LIN {X 0,Y 646.428,Z 1220.53,A -85,B 0,C 180,E1 5689.575,E2 5689.575} C_VEL
LIN {X 0,Y 649.933,Z 1168.755,A -85,B 0,C 180,E1 5694.149,E2 5694.149} C_VEL
LIN {X 0,Y 653.891,Z 1107.9,A -85,B 0,C 180,E1 5697.593,E2 5697.593} C_VEL
LIN {X 0,Y 656.115,Z 1042.809,A -85,B 0,C 180,E1 5699.566,E2 5699.566} C_VEL
LIN {X 0,Y 654.845,Z 982.129,A -85,B 0,C 180,E1 5700.484,E2 5700.484} C_VEL
LIN {X 0,Y 643.755,Z 957.34,A -85,B 0,C 180,E1 5701.335,E2 5701.335} C_VEL
LIN {X 0,Y 642.509,Z 948.94,A -85,B 0,C 180,E1 5701.958,E2 5701.958} C_VEL
LIN {X 0,Y 642.113,Z 948.94,A -85,B 0,C 180,E1 5710.571,E2 5710.571} C_VEL
LIN {X 0,Y 642.041,Z 948.94,A -85,B 0,C 180,E1 5718.158,E2 5718.158} C_VEL
LIN {X 0,Y 642.465,Z 950.207,A -85,B 0,C 180,E1 5726.456,E2 5726.456} C_VEL
LIN {X 0,Y 655.644,Z 990.43,A -85,B 0,C 180,E1 5727.732,E2 5727.732} C_VEL
LIN {X 0,Y 652.92,Z 1053.472,A -85,B 0,C 180,E1 5730.091,E2 5730.091} C_VEL
LIN {X 0,Y 649.225,Z 1112.123,A -85,B 0,C 180,E1 5733.83,E2 5733.83} C_VEL
LIN {X 0,Y 646.117,Z 1161.521,A -85,B 0,C 180,E1 5738.661,E2 5738.661} C_VEL
LIN {X 0,Y 644.175,Z 1198.737,A -85,B 0,C 180,E1 5744.292,E2 5744.292} C_VEL
LIN {X 0,Y 643.44,Z 1220.238,A -85,B 0,C 180,E1 5749.823,E2 5749.823} C_VEL
LIN {X 0,Y 643.165,Z 1229.44,A -85,B 0,C 180,E1 5755.275,E2 5755.275} C_VEL
LIN {X 0,Y 643.245,Z 1227.348,A -85,B 0,C 180,E1 5760.689,E2 5760.689} C_VEL
LIN {X 0,Y 643.485,Z 1212.675,A -85,B 0,C 180,E1 5766.446,E2 5766.446} C_VEL
LIN {X 0,Y 644.379,Z 1184.48,A -85,B 0,C 180,E1 5772.11,E2 5772.11} C_VEL
LIN {X 0,Y 646.945,Z 1142.6,A -85,B 0,C 180,E1 5777.367,E2 5777.367} C_VEL
LIN {X 0,Y 650.641,Z 1089.256,A -85,B 0,C 180,E1 5781.75,E2 5781.75} C_VEL
LIN {X 0,Y 654.328,Z 1028.717,A -85,B 0,C 180,E1 5784.935,E2 5784.935} C_VEL
LIN {X 0,Y 654.304,Z 979.292,A -85,B 0,C 180,E1 5786.611,E2 5786.611} C_VEL
LIN {X 0,Y 642.852,Z 948.94,A -85,B 0,C 180,E1 5787.961,E2 5787.961} C_VEL
LIN {X 0,Y 642.196,Z 948.94,A -85,B 0,C 180,E1 5797.622,E2 5797.622} C_VEL
LIN {X 0,Y 642.346,Z 948.94,A -85,B 0,C 180,E1 5806.13,E2 5806.13} C_VEL
LIN {X 0,Y 642.338,Z 948.94,A -85,B 0,C 180,E1 5814.631,E2 5814.631} C_VEL
LIN {X 0,Y 642.322,Z 948.94,A -85,B 0,C 180,E1 5822.535,E2 5822.535} C_VEL
LIN {X 0,Y 642.573,Z 948.94,A -85,B 0,C 180,E1 5829.943,E2 5829.943} C_VEL
LIN {X 0,Y 642.913,Z 950.765,A -85,B 0,C 180,E1 5832.35,E2 5832.35} C_VEL
LIN {X 0,Y 647.67,Z 983.205,A -85,B 0,C 180,E1 5832.85,E2 5832.85} C_VEL
LIN {X 0,Y 647.354,Z 1037.427,A -85,B 0,C 180,E1 5833.934,E2 5833.934} C_VEL
LIN {X 0,Y 645.952,Z 1082.258,A -85,B 0,C 180,E1 5836.208,E2 5836.208} C_VEL
LIN {X 0,Y 644.407,Z 1118.531,A -85,B 0,C 180,E1 5839.624,E2 5839.624} C_VEL
LIN {X 0,Y 643.495,Z 1142.198,A -85,B 0,C 180,E1 5843.876,E2 5843.876} C_VEL
LIN {X 0,Y 643.274,Z 1150.855,A -85,B 0,C 180,E1 5847.939,E2 5847.939} C_VEL
LIN {X 0,Y 643.428,Z 1148.022,A -85,B 0,C 180,E1 5851.994,E2 5851.994} C_VEL
LIN {X 0,Y 643.839,Z 1131.237,A -85,B 0,C 180,E1 5856.394,E2 5856.394} C_VEL
LIN {X 0,Y 644.983,Z 1101.717,A -85,B 0,C 180,E1 5860.128,E2 5860.128} C_VEL
LIN {X 0,Y 646.585,Z 1059.916,A -85,B 0,C 180,E1 5863.036,E2 5863.036} C_VEL
LIN {X 0,Y 647.882,Z 1011.403,A -85,B 0,C 180,E1 5864.667,E2 5864.667} C_VEL
LIN {X 0,Y 645.703,Z 960.583,A -85,B 0,C 180,E1 5865.371,E2 5865.371} C_VEL
LIN {X 0,Y 642.603,Z 948.94,A -85,B 0,C 180,E1 5865.721,E2 5865.721} C_VEL
LIN {X 0,Y 642.111,Z 948.94,A -85,B 0,C 180,E1 5872.911,E2 5872.911} C_VEL
LIN {X 0,Y 642.222,Z 948.94,A -85,B 0,C 180,E1 5880.488,E2 5880.488} C_VEL
LIN {X 0,Y 642.085,Z 948.94,A -85,B 0,C 180,E1 5888.728,E2 5888.728} C_VEL
LIN {X 0,Y 642.426,Z 948.94,A -85,B 0,C 180,E1 5896.035,E2 5896.035} C_VEL
LIN {X 0,Y 642.27,Z 948.94,A -85,B 0,C 180,E1 5904.605,E2 5904.605} C_VEL
LIN {X 0,Y 642.317,Z 948.94,A -85,B 0,C 180,E1 5912.547,E2 5912.547} C_VEL
LIN {X 0,Y 642.449,Z 948.94,A -85,B 0,C 180,E1 5919.953,E2 5919.953} C_VEL
LIN {X 0,Y 643.365,Z 948.94,A -85,B 0,C 180,E1 5928.419,E2 5928.419} C_VEL
LIN {X 0,Y 643.231,Z 948.94,A -85,B 0,C 180,E1 5937.958,E2 5937.958} C_VEL
LIN {X 0,Y 642.876,Z 948.94,A -85,B 0,C 180,E1 5946.085,E2 5946.085} C_VEL
LIN {X 0,Y 642.522,Z 948.94,A -85,B 0,C 180,E1 5954.348,E2 5954.348} C_VEL
LIN {X 0,Y 642.159,Z 948.94,A -85,B 0,C 180,E1 5962.94,E2 5962.94} C_VEL
LIN {X 0,Y 642.622,Z 948.94,A -85,B 0,C 180,E1 5970.548,E2 5970.548} C_VEL
LIN {X 0,Y 642.427,Z 948.94,A -85,B 0,C 180,E1 5979.155,E2 5979.155} C_VEL
LIN {X 0,Y 634.35,Z 948.94,A -85,B 0,C 180,E1 5982.271,E2 5982.271} C_VEL
LIN {X 0,Y 634.608,Z 948.94,A -85,B 0,C 180,E1 5990.994,E2 5990.994} C_VEL
LIN {X 0,Y 635.016,Z 950.715,A -85,B 0,C 180,E1 5996.544,E2 5996.544} C_VEL
LIN {X 0,Y 641.732,Z 974.807,A -85,B 0,C 180,E1 5998.37,E2 5998.37} C_VEL
LIN {X 0,Y 650.934,Z 992.589,A -85,B 0,C 180,E1 5999.107,E2 5999.107} C_VEL
LIN {X 0,Y 648.752,Z 1064.383,A -85,B 0,C 180,E1 6000.526,E2 6000.526} C_VEL
LIN {X 0,Y 645.117,Z 1130.85,A -85,B 0,C 180,E1 6003.225,E2 6003.225} C_VEL
LIN {X 0,Y 641.322,Z 1185.71,A -85,B 0,C 180,E1 6006.875,E2 6006.875} C_VEL
LIN {X 0,Y 638.039,Z 1233.34,A -85,B 0,C 180,E1 6011.693,E2 6011.693} C_VEL
LIN {X 0,Y 635.898,Z 1268.832,A -85,B 0,C 180,E1 6017.184,E2 6017.184} C_VEL
LIN {X 0,Y 635.105,Z 1289.609,A -85,B 0,C 180,E1 6022.548,E2 6022.548} C_VEL
LIN {X 0,Y 635.014,Z 1299.208,A -85,B 0,C 180,E1 6027.98,E2 6027.98} C_VEL
LIN {X 0,Y 634.95,Z 1297.779,A -85,B 0,C 180,E1 6033.459,E2 6033.459} C_VEL
LIN {X 0,Y 635.181,Z 1284.935,A -85,B 0,C 180,E1 6038.966,E2 6038.966} C_VEL
LIN {X 0,Y 636.236,Z 1259.453,A -85,B 0,C 180,E1 6044.536,E2 6044.536} C_VEL
LIN {X 0,Y 638.681,Z 1220.522,A -85,B 0,C 180,E1 6049.823,E2 6049.823} C_VEL
LIN {X 0,Y 642.5,Z 1168.755,A -85,B 0,C 180,E1 6054.447,E2 6054.447} C_VEL
LIN {X 0,Y 645.793,Z 1115.733,A -85,B 0,C 180,E1 6057.443,E2 6057.443} C_VEL
LIN {X 0,Y 648.319,Z 1043.871,A -85,B 0,C 180,E1 6059.711,E2 6059.711} C_VEL
LIN {X 0,Y 647.032,Z 984.427,A -85,B 0,C 180,E1 6060.682,E2 6060.682} C_VEL
LIN {X 0,Y 634.809,Z 952.48,A -85,B 0,C 180,E1 6061.606,E2 6061.606} C_VEL
LIN {X 0,Y 634.515,Z 948.94,A -85,B 0,C 180,E1 6061.902,E2 6061.902} C_VEL
LIN {X 0,Y 634.218,Z 948.94,A -85,B 0,C 180,E1 6069.387,E2 6069.387} C_VEL
LIN {X 0,Y 634.161,Z 948.94,A -85,B 0,C 180,E1 6077.009,E2 6077.009} C_VEL
LIN {X 0,Y 634.329,Z 948.94,A -85,B 0,C 180,E1 6086.148,E2 6086.148} C_VEL
LIN {X 0,Y 648.172,Z 992.693,A -85,B 0,C 180,E1 6087.529,E2 6087.529} C_VEL
LIN {X 0,Y 645.371,Z 1056.755,A -85,B 0,C 180,E1 6089.964,E2 6089.964} C_VEL
LIN {X 0,Y 641.651,Z 1112.722,A -85,B 0,C 180,E1 6093.591,E2 6093.591} C_VEL
LIN {X 0,Y 638.341,Z 1161.181,A -85,B 0,C 180,E1 6098.388,E2 6098.388} C_VEL
LIN {X 0,Y 636.325,Z 1198.539,A -85,B 0,C 180,E1 6104.093,E2 6104.093} C_VEL
LIN {X 0,Y 635.515,Z 1220.127,A -85,B 0,C 180,E1 6109.695,E2 6109.695} C_VEL
LIN {X 0,Y 635.167,Z 1229.413,A -85,B 0,C 180,E1 6115.216,E2 6115.216} C_VEL
LIN {X 0,Y 635.239,Z 1227.405,A -85,B 0,C 180,E1 6120.698,E2 6120.698} C_VEL
LIN {X 0,Y 635.5,Z 1212.876,A -85,B 0,C 180,E1 6126.508,E2 6126.508} C_VEL
LIN {X 0,Y 636.492,Z 1184.73,A -85,B 0,C 180,E1 6132.262,E2 6132.262} C_VEL
LIN {X 0,Y 639.204,Z 1143.404,A -85,B 0,C 180,E1 6137.542,E2 6137.542} C_VEL
LIN {X 0,Y 643.18,Z 1089.823,A -85,B 0,C 180,E1 6142.015,E2 6142.015} C_VEL
LIN {X 0,Y 647.176,Z 1028.483,A -85,B 0,C 180,E1 6145.268,E2 6145.268} C_VEL
LIN {X 0,Y 647.023,Z 981.257,A -85,B 0,C 180,E1 6146.902,E2 6146.902} C_VEL
LIN {X 0,Y 634.781,Z 948.94,A -85,B 0,C 180,E1 6148.335,E2 6148.335} C_VEL
LIN {X 0,Y 634.2,Z 948.94,A -85,B 0,C 180,E1 6157.627,E2 6157.627} C_VEL
LIN {X 0,Y 634.2,Z 948.94,A -85,B 0,C 180,E1 6166.966,E2 6166.966} C_VEL
LIN {X 0,Y 634.188,Z 948.94,A -85,B 0,C 180,E1 6175.749,E2 6175.749} C_VEL
LIN {X 0,Y 634.257,Z 948.94,A -85,B 0,C 180,E1 6183.848,E2 6183.848} C_VEL
LIN {X 0,Y 634.715,Z 950.059,A -85,B 0,C 180,E1 6192.111,E2 6192.111} C_VEL
LIN {X 0,Y 640.019,Z 982.816,A -85,B 0,C 180,E1 6192.638,E2 6192.638} C_VEL
LIN {X 0,Y 639.702,Z 1038.025,A -85,B 0,C 180,E1 6193.739,E2 6193.739} C_VEL
LIN {X 0,Y 638.223,Z 1083.011,A -85,B 0,C 180,E1 6196.037,E2 6196.037} C_VEL
LIN {X 0,Y 636.603,Z 1119.38,A -85,B 0,C 180,E1 6199.495,E2 6199.495} C_VEL
LIN {X 0,Y 635.609,Z 1143.099,A -85,B 0,C 180,E1 6203.799,E2 6203.799} C_VEL
LIN {X 0,Y 635.36,Z 1151.796,A -85,B 0,C 180,E1 6207.913,E2 6207.913} C_VEL
LIN {X 0,Y 635.503,Z 1149.001,A -85,B 0,C 180,E1 6212.019,E2 6212.019} C_VEL
LIN {X 0,Y 635.962,Z 1132.256,A -85,B 0,C 180,E1 6216.473,E2 6216.473} C_VEL
LIN {X 0,Y 637.199,Z 1102.796,A -85,B 0,C 180,E1 6220.253,E2 6220.253} C_VEL
LIN {X 0,Y 638.869,Z 1062.061,A -85,B 0,C 180,E1 6223.144,E2 6223.144} C_VEL
LIN {X 0,Y 640.219,Z 1013.84,A -85,B 0,C 180,E1 6224.829,E2 6224.829} C_VEL
LIN {X 0,Y 637.967,Z 961.761,A -85,B 0,C 180,E1 6225.571,E2 6225.571} C_VEL
LIN {X 0,Y 634.577,Z 948.94,A -85,B 0,C 180,E1 6225.925,E2 6225.925} C_VEL
LIN {X 0,Y 634.047,Z 948.94,A -85,B 0,C 180,E1 6233.219,E2 6233.219} C_VEL
LIN {X 0,Y 634.111,Z 948.94,A -85,B 0,C 180,E1 6240.921,E2 6240.921} C_VEL
LIN {X 0,Y 634.014,Z 948.94,A -85,B 0,C 180,E1 6249.315,E2 6249.315} C_VEL
LIN {X 0,Y 634.267,Z 948.94,A -85,B 0,C 180,E1 6256.981,E2 6256.981} C_VEL
LIN {X 0,Y 634.154,Z 948.94,A -85,B 0,C 180,E1 6265.758,E2 6265.758} C_VEL
LIN {X 0,Y 634.271,Z 948.94,A -85,B 0,C 180,E1 6273.709,E2 6273.709} C_VEL
LIN {X 0,Y 634.326,Z 948.94,A -85,B 0,C 180,E1 6281.14,E2 6281.14} C_VEL
LIN {X 0,Y 635.376,Z 948.94,A -85,B 0,C 180,E1 6288.271,E2 6288.271} C_VEL
LIN {X 0,Y 635.231,Z 948.94,A -85,B 0,C 180,E1 6297.933,E2 6297.933} C_VEL
LIN {X 0,Y 634.835,Z 948.94,A -85,B 0,C 180,E1 6306.163,E2 6306.163} C_VEL
LIN {X 0,Y 634.471,Z 948.94,A -85,B 0,C 180,E1 6314.552,E2 6314.552} C_VEL
LIN {X 0,Y 634.146,Z 948.94,A -85,B 0,C 180,E1 6322.991,E2 6322.991} C_VEL
LIN {X 0,Y 634.596,Z 948.94,A -85,B 0,C 180,E1 6330.93,E2 6330.93} C_VEL
LIN {X 0,Y 634.449,Z 948.94,A -85,B 0,C 180,E1 6339.326,E2 6339.326} C_VEL
LIN {X 0,Y 634.35,Z 948.94,A -85,B 0,C 180,E1 6342.271,E2 6342.271} C_VEL
LIN {X 0,Y 626.079,Z 948.94,A -85,B 0,C 180,E1 6345.419,E2 6345.419} C_VEL
LIN {X 0,Y 626.58,Z 948.94,A -85,B 0,C 180,E1 6354.219,E2 6354.219} C_VEL
LIN {X 0,Y 626.844,Z 950.065,A -85,B 0,C 180,E1 6356.109,E2 6356.109} C_VEL
LIN {X 0,Y 632.967,Z 973.261,A -85,B 0,C 180,E1 6357.845,E2 6357.845} C_VEL
LIN {X 0,Y 644.086,Z 995.648,A -85,B 0,C 180,E1 6358.778,E2 6358.778} C_VEL
LIN {X 0,Y 641.476,Z 1066.107,A -85,B 0,C 180,E1 6360.256,E2 6360.256} C_VEL
LIN {X 0,Y 637.418,Z 1134.053,A -85,B 0,C 180,E1 6363.134,E2 6363.134} C_VEL
LIN {X 0,Y 633.274,Z 1192.218,A -85,B 0,C 180,E1 6367.127,E2 6367.127} C_VEL
LIN {X 0,Y 629.723,Z 1239.53,A -85,B 0,C 180,E1 6372.255,E2 6372.255} C_VEL
LIN {X 0,Y 627.749,Z 1272.634,A -85,B 0,C 180,E1 6377.825,E2 6377.825} C_VEL
LIN {X 0,Y 627.021,Z 1291.733,A -85,B 0,C 180,E1 6383.228,E2 6383.228} C_VEL
LIN {X 0,Y 627.039,Z 1299.203,A -85,B 0,C 180,E1 6387.954,E2 6387.954} C_VEL
LIN {X 0,Y 626.947,Z 1297.781,A -85,B 0,C 180,E1 6393.503,E2 6393.503} C_VEL
LIN {X 0,Y 627.192,Z 1284.932,A -85,B 0,C 180,E1 6399.082,E2 6399.082} C_VEL
LIN {X 0,Y 628.329,Z 1259.448,A -85,B 0,C 180,E1 6404.723,E2 6404.723} C_VEL
LIN {X 0,Y 630.95,Z 1220.807,A -85,B 0,C 180,E1 6410.041,E2 6410.041} C_VEL
LIN {X 0,Y 634.709,Z 1171.858,A -85,B 0,C 180,E1 6414.484,E2 6414.484} C_VEL
LIN {X 0,Y 638.039,Z 1111.305,A -85,B 0,C 180,E1 6417.73,E2 6417.73} C_VEL
LIN {X 0,Y 640.739,Z 1039.901,A -85,B 0,C 180,E1 6419.968,E2 6419.968} C_VEL
LIN {X 0,Y 639.776,Z 987.462,A -85,B 0,C 180,E1 6420.86,E2 6420.86} C_VEL
LIN {X 0,Y 626.799,Z 952.316,A -85,B 0,C 180,E1 6421.684,E2 6421.684} C_VEL
LIN {X 0,Y 626.474,Z 948.94,A -85,B 0,C 180,E1 6422.081,E2 6422.081} C_VEL
LIN {X 0,Y 626.1,Z 948.94,A -85,B 0,C 180,E1 6430.236,E2 6430.236} C_VEL
LIN {X 0,Y 625.956,Z 948.94,A -85,B 0,C 180,E1 6438.197,E2 6438.197} C_VEL
LIN {X 0,Y 626.473,Z 950.495,A -85,B 0,C 180,E1 6445.907,E2 6445.907} C_VEL
LIN {X 0,Y 640.707,Z 994.789,A -85,B 0,C 180,E1 6447.317,E2 6447.317} C_VEL
LIN {X 0,Y 637.846,Z 1058.518,A -85,B 0,C 180,E1 6449.772,E2 6449.772} C_VEL
LIN {X 0,Y 634.019,Z 1114.463,A -85,B 0,C 180,E1 6453.44,E2 6453.44} C_VEL
LIN {X 0,Y 630.506,Z 1162.288,A -85,B 0,C 180,E1 6458.292,E2 6458.292} C_VEL
LIN {X 0,Y 628.438,Z 1198.34,A -85,B 0,C 180,E1 6463.888,E2 6463.888} C_VEL
LIN {X 0,Y 627.556,Z 1220.016,A -85,B 0,C 180,E1 6469.563,E2 6469.563} C_VEL
LIN {X 0,Y 627.179,Z 1229.387,A -85,B 0,C 180,E1 6475.155,E2 6475.155} C_VEL
LIN {X 0,Y 627.233,Z 1227.462,A -85,B 0,C 180,E1 6480.707,E2 6480.707} C_VEL
LIN {X 0,Y 627.527,Z 1214.163,A -85,B 0,C 180,E1 6486.262,E2 6486.262} C_VEL
LIN {X 0,Y 628.523,Z 1186.703,A -85,B 0,C 180,E1 6492.145,E2 6492.145} C_VEL
LIN {X 0,Y 631.343,Z 1146.137,A -85,B 0,C 180,E1 6497.502,E2 6497.502} C_VEL
LIN {X 0,Y 635.583,Z 1092.946,A -85,B 0,C 180,E1 6502.108,E2 6502.108} C_VEL
LIN {X 0,Y 639.779,Z 1032.03,A -85,B 0,C 180,E1 6505.451,E2 6505.451} C_VEL
LIN {X 0,Y 639.99,Z 983.789,A -85,B 0,C 180,E1 6507.174,E2 6507.174} C_VEL
LIN {X 0,Y 626.682,Z 948.94,A -85,B 0,C 180,E1 6508.707,E2 6508.707} C_VEL
LIN {X 0,Y 626.098,Z 948.94,A -85,B 0,C 180,E1 6518.201,E2 6518.201} C_VEL
LIN {X 0,Y 626.182,Z 948.94,A -85,B 0,C 180,E1 6526.278,E2 6526.278} C_VEL
LIN {X 0,Y 626.19,Z 948.94,A -85,B 0,C 180,E1 6535.249,E2 6535.249} C_VEL
LIN {X 0,Y 626.255,Z 948.94,A -85,B 0,C 180,E1 6543.333,E2 6543.333} C_VEL
LIN {X 0,Y 626.611,Z 948.94,A -85,B 0,C 180,E1 6551.857,E2 6551.857} C_VEL
LIN {X 0,Y 632.346,Z 981.432,A -85,B 0,C 180,E1 6552.409,E2 6552.409} C_VEL
LIN {X 0,Y 632.084,Z 1037.191,A -85,B 0,C 180,E1 6553.492,E2 6553.492} C_VEL
LIN {X 0,Y 630.585,Z 1082.539,A -85,B 0,C 180,E1 6555.776,E2 6555.776} C_VEL
LIN {X 0,Y 628.926,Z 1118.829,A -85,B 0,C 180,E1 6559.189,E2 6559.189} C_VEL
LIN {X 0,Y 627.934,Z 1142.695,A -85,B 0,C 180,E1 6563.375,E2 6563.375} C_VEL
LIN {X 0,Y 627.434,Z 1152.737,A -85,B 0,C 180,E1 6567.887,E2 6567.887} C_VEL
LIN {X 0,Y 627.592,Z 1149.978,A -85,B 0,C 180,E1 6572.044,E2 6572.044} C_VEL
LIN {X 0,Y 628.079,Z 1133.276,A -85,B 0,C 180,E1 6576.555,E2 6576.555} C_VEL
LIN {X 0,Y 629.416,Z 1103.874,A -85,B 0,C 180,E1 6580.381,E2 6580.381} C_VEL
LIN {X 0,Y 631.176,Z 1062.572,A -85,B 0,C 180,E1 6583.343,E2 6583.343} C_VEL
LIN {X 0,Y 632.576,Z 1015.377,A -85,B 0,C 180,E1 6585.012,E2 6585.012} C_VEL
LIN {X 0,Y 630.22,Z 962.615,A -85,B 0,C 180,E1 6585.781,E2 6585.781} C_VEL
LIN {X 0,Y 626.541,Z 948.94,A -85,B 0,C 180,E1 6586.134,E2 6586.134} C_VEL
LIN {X 0,Y 625.957,Z 948.94,A -85,B 0,C 180,E1 6594.56,E2 6594.56} C_VEL
LIN {X 0,Y 626.037,Z 948.94,A -85,B 0,C 180,E1 6601.364,E2 6601.364} C_VEL
LIN {X 0,Y 625.922,Z 948.94,A -85,B 0,C 180,E1 6609.924,E2 6609.924} C_VEL
LIN {X 0,Y 626.144,Z 948.94,A -85,B 0,C 180,E1 6618.175,E2 6618.175} C_VEL
LIN {X 0,Y 626.16,Z 948.94,A -85,B 0,C 180,E1 6626.932,E2 6626.932} C_VEL
LIN {X 0,Y 626.41,Z 948.94,A -85,B 0,C 180,E1 6635.191,E2 6635.191} C_VEL
LIN {X 0,Y 626.674,Z 948.94,A -85,B 0,C 180,E1 6643.813,E2 6643.813} C_VEL
LIN {X 0,Y 626.802,Z 948.94,A -85,B 0,C 180,E1 6650.93,E2 6650.93} C_VEL
LIN {X 0,Y 627.241,Z 948.94,A -85,B 0,C 180,E1 6657.906,E2 6657.906} C_VEL
LIN {X 0,Y 626.804,Z 948.94,A -85,B 0,C 180,E1 6666.242,E2 6666.242} C_VEL
LIN {X 0,Y 626.438,Z 948.94,A -85,B 0,C 180,E1 6674.724,E2 6674.724} C_VEL
LIN {X 0,Y 626.313,Z 948.94,A -85,B 0,C 180,E1 6682.048,E2 6682.048} C_VEL
LIN {X 0,Y 626.574,Z 948.94,A -85,B 0,C 180,E1 6691.371,E2 6691.371} C_VEL
LIN {X 0,Y 626.387,Z 948.94,A -85,B 0,C 180,E1 6699.933,E2 6699.933} C_VEL
LIN {X 0,Y 626.079,Z 948.94,A -85,B 0,C 180,E1 6705.419,E2 6705.419} C_VEL
LIN {X 0,Y 618.251,Z 948.94,A -85,B 0,C 180,E1 6708.612,E2 6708.612} C_VEL
LIN {X 0,Y 618.915,Z 950.77,A -85,B 0,C 180,E1 6715.779,E2 6715.779} C_VEL
LIN {X 0,Y 624.625,Z 971.408,A -85,B 0,C 180,E1 6717.323,E2 6717.323} C_VEL
LIN {X 0,Y 637.204,Z 1000.02,A -85,B 0,C 180,E1 6718.456,E2 6718.456} C_VEL
LIN {X 0,Y 634.063,Z 1071.337,A -85,B 0,C 180,E1 6720.099,E2 6720.099} C_VEL
LIN {X 0,Y 629.657,Z 1138.218,A -85,B 0,C 180,E1 6723.096,E2 6723.096} C_VEL
LIN {X 0,Y 625.202,Z 1196.624,A -85,B 0,C 180,E1 6727.288,E2 6727.288} C_VEL
LIN {X 0,Y 621.925,Z 1239.976,A -85,B 0,C 180,E1 6732.085,E2 6732.085} C_VEL
LIN {X 0,Y 619.805,Z 1272.628,A -85,B 0,C 180,E1 6737.667,E2 6737.667} C_VEL
LIN {X 0,Y 619.05,Z 1291.611,A -85,B 0,C 180,E1 6743.096,E2 6743.096} C_VEL
LIN {X 0,Y 619.045,Z 1299.198,A -85,B 0,C 180,E1 6747.928,E2 6747.928} C_VEL
LIN {X 0,Y 618.943,Z 1297.777,A -85,B 0,C 180,E1 6753.548,E2 6753.548} C_VEL
LIN {X 0,Y 619.237,Z 1284.93,A -85,B 0,C 180,E1 6759.199,E2 6759.199} C_VEL
LIN {X 0,Y 620.438,Z 1259.444,A -85,B 0,C 180,E1 6764.915,E2 6764.915} C_VEL
LIN {X 0,Y 623.332,Z 1219.873,A -85,B 0,C 180,E1 6770.408,E2 6770.408} C_VEL
LIN {X 0,Y 626.61,Z 1175.783,A -85,B 0,C 180,E1 6774.299,E2 6774.299} C_VEL
LIN {X 0,Y 630.082,Z 1112.795,A -85,B 0,C 180,E1 6777.787,E2 6777.787} C_VEL
LIN {X 0,Y 633.027,Z 1038.375,A -85,B 0,C 180,E1 6780.182,E2 6780.182} C_VEL
LIN {X 0,Y 632.053,Z 989.56,A -85,B 0,C 180,E1 6781.066,E2 6781.066} C_VEL
LIN {X 0,Y 619.47,Z 954.539,A -85,B 0,C 180,E1 6781.911,E2 6781.911} C_VEL
LIN {X 0,Y 618.455,Z 948.94,A -85,B 0,C 180,E1 6782.172,E2 6782.172} C_VEL
LIN {X 0,Y 618.077,Z 948.94,A -85,B 0,C 180,E1 6790.627,E2 6790.627} C_VEL
LIN {X 0,Y 617.935,Z 948.94,A -85,B 0,C 180,E1 6798.547,E2 6798.547} C_VEL
LIN {X 0,Y 618.365,Z 949.669,A -85,B 0,C 180,E1 6805.599,E2 6805.599} C_VEL
LIN {X 0,Y 633.261,Z 997.105,A -85,B 0,C 180,E1 6807.107,E2 6807.107} C_VEL
LIN {X 0,Y 630.352,Z 1059.6,A -85,B 0,C 180,E1 6809.541,E2 6809.541} C_VEL
LIN {X 0,Y 626.359,Z 1116.16,A -85,B 0,C 180,E1 6813.292,E2 6813.292} C_VEL
LIN {X 0,Y 622.674,Z 1163.395,A -85,B 0,C 180,E1 6818.193,E2 6818.193} C_VEL
LIN {X 0,Y 620.378,Z 1199.846,A -85,B 0,C 180,E1 6824.038,E2 6824.038} C_VEL
LIN {X 0,Y 619.335,Z 1221.829,A -85,B 0,C 180,E1 6830.136,E2 6830.136} C_VEL
LIN {X 0,Y 619.179,Z 1229.36,A -85,B 0,C 180,E1 6835.092,E2 6835.092} C_VEL
LIN {X 0,Y 619.228,Z 1227.518,A -85,B 0,C 180,E1 6840.716,E2 6840.716} C_VEL
LIN {X 0,Y 619.526,Z 1212.665,A -85,B 0,C 180,E1 6846.815,E2 6846.815} C_VEL
LIN {X 0,Y 620.684,Z 1185.427,A -85,B 0,C 180,E1 6852.549,E2 6852.549} C_VEL
LIN {X 0,Y 623.724,Z 1144.944,A -85,B 0,C 180,E1 6857.901,E2 6857.901} C_VEL
LIN {X 0,Y 628.258,Z 1092.305,A -85,B 0,C 180,E1 6862.473,E2 6862.473} C_VEL
LIN {X 0,Y 632.699,Z 1031.07,A -85,B 0,C 180,E1 6865.83,E2 6865.83} C_VEL
LIN {X 0,Y 632.951,Z 986.353,A -85,B 0,C 180,E1 6867.452,E2 6867.452} C_VEL
LIN {X 0,Y 618.528,Z 948.94,A -85,B 0,C 180,E1 6869.237,E2 6869.237} C_VEL
LIN {X 0,Y 618.144,Z 948.94,A -85,B 0,C 180,E1 6877.029,E2 6877.029} C_VEL
LIN {X 0,Y 618.174,Z 948.94,A -85,B 0,C 180,E1 6886.432,E2 6886.432} C_VEL
LIN {X 0,Y 618.192,Z 948.94,A -85,B 0,C 180,E1 6895.36,E2 6895.36} C_VEL
LIN {X 0,Y 618.254,Z 948.94,A -85,B 0,C 180,E1 6903.677,E2 6903.677} C_VEL
LIN {X 0,Y 618.771,Z 950.635,A -85,B 0,C 180,E1 6911.648,E2 6911.648} C_VEL
LIN {X 0,Y 624.724,Z 982.863,A -85,B 0,C 180,E1 6912.209,E2 6912.209} C_VEL
LIN {X 0,Y 624.437,Z 1038.371,A -85,B 0,C 180,E1 6913.308,E2 6913.308} C_VEL
LIN {X 0,Y 622.867,Z 1083.29,A -85,B 0,C 180,E1 6915.596,E2 6915.596} C_VEL
LIN {X 0,Y 621.131,Z 1119.667,A -85,B 0,C 180,E1 6919.052,E2 6919.052} C_VEL
LIN {X 0,Y 620.039,Z 1143.673,A -85,B 0,C 180,E1 6923.311,E2 6923.311} C_VEL
LIN {X 0,Y 619.52,Z 1153.678,A -85,B 0,C 180,E1 6927.86,E2 6927.86} C_VEL
LIN {X 0,Y 619.665,Z 1150.957,A -85,B 0,C 180,E1 6932.07,E2 6932.07} C_VEL
LIN {X 0,Y 620.206,Z 1134.293,A -85,B 0,C 180,E1 6936.638,E2 6936.638} C_VEL
LIN {X 0,Y 621.646,Z 1104.95,A -85,B 0,C 180,E1 6940.513,E2 6940.513} C_VEL
LIN {X 0,Y 623.493,Z 1063.739,A -85,B 0,C 180,E1 6943.51,E2 6943.51} C_VEL
LIN {X 0,Y 624.931,Z 1016.15,A -85,B 0,C 180,E1 6945.215,E2 6945.215} C_VEL
LIN {X 0,Y 622.549,Z 963.94,A -85,B 0,C 180,E1 6945.987,E2 6945.987} C_VEL
LIN {X 0,Y 618.515,Z 948.94,A -85,B 0,C 180,E1 6946.35,E2 6946.35} C_VEL
LIN {X 0,Y 617.962,Z 948.94,A -85,B 0,C 180,E1 6953.861,E2 6953.861} C_VEL
LIN {X 0,Y 617.955,Z 948.94,A -85,B 0,C 180,E1 6962.046,E2 6962.046} C_VEL
LIN {X 0,Y 617.897,Z 948.94,A -85,B 0,C 180,E1 6970.55,E2 6970.55} C_VEL
LIN {X 0,Y 618.146,Z 948.94,A -85,B 0,C 180,E1 6978.42,E2 6978.42} C_VEL
LIN {X 0,Y 618.157,Z 948.94,A -85,B 0,C 180,E1 6986.448,E2 6986.448} C_VEL
LIN {X 0,Y 618.303,Z 948.94,A -85,B 0,C 180,E1 6994.543,E2 6994.543} C_VEL
LIN {X 0,Y 618.637,Z 948.94,A -85,B 0,C 180,E1 7003.597,E2 7003.597} C_VEL
LIN {X 0,Y 618.846,Z 948.94,A -85,B 0,C 180,E1 7010.813,E2 7010.813} C_VEL
LIN {X 0,Y 619.24,Z 948.94,A -85,B 0,C 180,E1 7017.879,E2 7017.879} C_VEL
LIN {X 0,Y 618.58,Z 948.94,A -85,B 0,C 180,E1 7026.886,E2 7026.886} C_VEL
LIN {X 0,Y 618.388,Z 948.94,A -85,B 0,C 180,E1 7034.92,E2 7034.92} C_VEL
LIN {X 0,Y 618.1,Z 948.94,A -85,B 0,C 180,E1 7043.086,E2 7043.086} C_VEL
LIN {X 0,Y 618.517,Z 948.94,A -85,B 0,C 180,E1 7051.827,E2 7051.827} C_VEL
LIN {X 0,Y 618.376,Z 948.94,A -85,B 0,C 180,E1 7060.557,E2 7060.557} C_VEL
LIN {X 0,Y 618.251,Z 948.94,A -85,B 0,C 180,E1 7068.612,E2 7068.612} C_VEL
LIN {X 0,Y 610.423,Z 948.94,A -85,B 0,C 180,E1 7071.854,E2 7071.854} C_VEL
LIN {X 0,Y 610.931,Z 950.999,A -85,B 0,C 180,E1 7075.398,E2 7075.398} C_VEL
LIN {X 0,Y 616.423,Z 969.525,A -85,B 0,C 180,E1 7076.791,E2 7076.791} C_VEL
LIN {X 0,Y 630.273,Z 1003.491,A -85,B 0,C 180,E1 7078.131,E2 7078.131} C_VEL
LIN {X 0,Y 626.759,Z 1074.429,A -85,B 0,C 180,E1 7079.874,E2 7079.874} C_VEL
LIN {X 0,Y 621.981,Z 1140.429,A -85,B 0,C 180,E1 7082.959,E2 7082.959} C_VEL
LIN {X 0,Y 617.26,Z 1198.745,A -85,B 0,C 180,E1 7087.284,E2 7087.284} C_VEL
LIN {X 0,Y 613.915,Z 1242.494,A -85,B 0,C 180,E1 7092.209,E2 7092.209} C_VEL
LIN {X 0,Y 611.772,Z 1274.278,A -85,B 0,C 180,E1 7097.866,E2 7097.866} C_VEL
LIN {X 0,Y 610.988,Z 1292.968,A -85,B 0,C 180,E1 7103.619,E2 7103.619} C_VEL
LIN {X 0,Y 610.897,Z 1299.825,A -85,B 0,C 180,E1 7109.324,E2 7109.324} C_VEL
LIN {X 0,Y 611.028,Z 1295.691,A -85,B 0,C 180,E1 7115.021,E2 7115.021} C_VEL
LIN {X 0,Y 611.898,Z 1277.935,A -85,B 0,C 180,E1 7121.247,E2 7121.247} C_VEL
LIN {X 0,Y 614,Z 1245.824,A -85,B 0,C 180,E1 7127.286,E2 7127.286} C_VEL
LIN {X 0,Y 616.497,Z 1208.513,A -85,B 0,C 180,E1 7131.702,E2 7131.702} C_VEL
LIN {X 0,Y 619.944,Z 1153.925,A -85,B 0,C 180,E1 7135.787,E2 7135.787} C_VEL
LIN {X 0,Y 623.434,Z 1085.707,A -85,B 0,C 180,E1 7138.975,E2 7138.975} C_VEL
LIN {X 0,Y 626.162,Z 1007.58,A -85,B 0,C 180,E1 7140.976,E2 7140.976} C_VEL
LIN {X 0,Y 623.591,Z 990.18,A -85,B 0,C 180,E1 7141.323,E2 7141.323} C_VEL
LIN {X 0,Y 610.42,Z 948.94,A -85,B 0,C 180,E1 7142.345,E2 7142.345} C_VEL
LIN {X 0,Y 610.079,Z 948.94,A -85,B 0,C 180,E1 7151.275,E2 7151.275} C_VEL
LIN {X 0,Y 609.921,Z 948.94,A -85,B 0,C 180,E1 7159.406,E2 7159.406} C_VEL
LIN {X 0,Y 610.447,Z 950.512,A -85,B 0,C 180,E1 7165.306,E2 7165.306} C_VEL
LIN {X 0,Y 625.776,Z 1000.068,A -85,B 0,C 180,E1 7166.908,E2 7166.908} C_VEL
LIN {X 0,Y 622.717,Z 1063.063,A -85,B 0,C 180,E1 7169.432,E2 7169.432} C_VEL
LIN {X 0,Y 618.644,Z 1118.961,A -85,B 0,C 180,E1 7173.236,E2 7173.236} C_VEL
LIN {X 0,Y 614.856,Z 1164.474,A -85,B 0,C 180,E1 7178.086,E2 7178.086} C_VEL
LIN {X 0,Y 612.499,Z 1199.646,A -85,B 0,C 180,E1 7183.827,E2 7183.827} C_VEL
LIN {X 0,Y 611.382,Z 1221.73,A -85,B 0,C 180,E1 7190.006,E2 7190.006} C_VEL
LIN {X 0,Y 611.176,Z 1229.325,A -85,B 0,C 180,E1 7195.028,E2 7195.028} C_VEL
LIN {X 0,Y 611.224,Z 1227.573,A -85,B 0,C 180,E1 7200.725,E2 7200.725} C_VEL
LIN {X 0,Y 611.536,Z 1213.247,A -85,B 0,C 180,E1 7206.773,E2 7206.773} C_VEL
LIN {X 0,Y 612.83,Z 1185.677,A -85,B 0,C 180,E1 7212.712,E2 7212.712} C_VEL
LIN {X 0,Y 616.166,Z 1143.96,A -85,B 0,C 180,E1 7218.307,E2 7218.307} C_VEL
LIN {X 0,Y 621.042,Z 1090.403,A -85,B 0,C 180,E1 7222.939,E2 7222.939} C_VEL
LIN {X 0,Y 625.784,Z 1028.143,A -85,B 0,C 180,E1 7226.301,E2 7226.301} C_VEL
LIN {X 0,Y 625.691,Z 988.359,A -85,B 0,C 180,E1 7227.756,E2 7227.756} C_VEL
LIN {X 0,Y 610.39,Z 948.94,A -85,B 0,C 180,E1 7229.635,E2 7229.635} C_VEL
LIN {X 0,Y 609.985,Z 948.94,A -85,B 0,C 180,E1 7238.359,E2 7238.359} C_VEL
LIN {X 0,Y 610.144,Z 948.94,A -85,B 0,C 180,E1 7247.23,E2 7247.23} C_VEL
LIN {X 0,Y 610.157,Z 948.94,A -85,B 0,C 180,E1 7255.936,E2 7255.936} C_VEL
LIN {X 0,Y 610.264,Z 948.94,A -85,B 0,C 180,E1 7264.17,E2 7264.17} C_VEL
LIN {X 0,Y 610.807,Z 950.847,A -85,B 0,C 180,E1 7271.404,E2 7271.404} C_VEL
LIN {X 0,Y 617.069,Z 981.887,A -85,B 0,C 180,E1 7271.971,E2 7271.971} C_VEL
LIN {X 0,Y 616.827,Z 1038.25,A -85,B 0,C 180,E1 7273.072,E2 7273.072} C_VEL
LIN {X 0,Y 615.178,Z 1084.052,A -85,B 0,C 180,E1 7275.412,E2 7275.412} C_VEL
LIN {X 0,Y 613.342,Z 1120.506,A -85,B 0,C 180,E1 7278.911,E2 7278.911} C_VEL
LIN {X 0,Y 612.256,Z 1143.851,A -85,B 0,C 180,E1 7283.033,E2 7283.033} C_VEL
LIN {X 0,Y 611.597,Z 1154.619,A -85,B 0,C 180,E1 7287.832,E2 7287.832} C_VEL
LIN {X 0,Y 611.728,Z 1151.938,A -85,B 0,C 180,E1 7292.097,E2 7292.097} C_VEL
LIN {X 0,Y 612.342,Z 1135.601,A -85,B 0,C 180,E1 7296.668,E2 7296.668} C_VEL
LIN {X 0,Y 613.872,Z 1106.025,A -85,B 0,C 180,E1 7300.647,E2 7300.647} C_VEL
LIN {X 0,Y 615.805,Z 1064.885,A -85,B 0,C 180,E1 7303.682,E2 7303.682} C_VEL
LIN {X 0,Y 617.274,Z 1017.605,A -85,B 0,C 180,E1 7305.409,E2 7305.409} C_VEL
LIN {X 0,Y 615.138,Z 966.152,A -85,B 0,C 180,E1 7306.179,E2 7306.179} C_VEL
LIN {X 0,Y 610.488,Z 948.94,A -85,B 0,C 180,E1 7306.571,E2 7306.571} C_VEL
LIN {X 0,Y 609.915,Z 948.94,A -85,B 0,C 180,E1 7314.692,E2 7314.692} C_VEL
LIN {X 0,Y 609.942,Z 948.94,A -85,B 0,C 180,E1 7322.29,E2 7322.29} C_VEL
LIN {X 0,Y 609.912,Z 948.94,A -85,B 0,C 180,E1 7331.195,E2 7331.195} C_VEL
LIN {X 0,Y 610.117,Z 948.94,A -85,B 0,C 180,E1 7339.277,E2 7339.277} C_VEL
LIN {X 0,Y 610.218,Z 948.94,A -85,B 0,C 180,E1 7347.655,E2 7347.655} C_VEL
LIN {X 0,Y 610.39,Z 948.94,A -85,B 0,C 180,E1 7355.762,E2 7355.762} C_VEL
LIN {X 0,Y 610.898,Z 948.94,A -85,B 0,C 180,E1 7364.863,E2 7364.863} C_VEL
LIN {X 0,Y 610.475,Z 948.94,A -85,B 0,C 180,E1 7372.126,E2 7372.126} C_VEL
LIN {X 0,Y 610.627,Z 948.94,A -85,B 0,C 180,E1 7379.274,E2 7379.274} C_VEL
LIN {X 0,Y 610.731,Z 948.94,A -85,B 0,C 180,E1 7386.407,E2 7386.407} C_VEL
LIN {X 0,Y 610.329,Z 948.94,A -85,B 0,C 180,E1 7395.122,E2 7395.122} C_VEL
LIN {X 0,Y 610.169,Z 948.94,A -85,B 0,C 180,E1 7402.664,E2 7402.664} C_VEL
LIN {X 0,Y 610.481,Z 948.94,A -85,B 0,C 180,E1 7411.037,E2 7411.037} C_VEL
LIN {X 0,Y 610.338,Z 948.94,A -85,B 0,C 180,E1 7419.338,E2 7419.338} C_VEL
LIN {X 0,Y 610.278,Z 948.94,A -85,B 0,C 180,E1 7428.835,E2 7428.835} C_VEL
LIN {X 0,Y 610.423,Z 948.94,A -85,B 0,C 180,E1 7431.854,E2 7431.854} C_VEL
LIN {X 0,Y 602.479,Z 948.94,A -85,B 0,C 180,E1 7433.992,E2 7433.992} C_VEL
LIN {X 0,Y 602.677,Z 950.167,A -85,B 0,C 180,E1 7434.91,E2 7434.91} C_VEL
LIN {X 0,Y 608.326,Z 968.385,A -85,B 0,C 180,E1 7436.26,E2 7436.26} C_VEL
LIN {X 0,Y 623.414,Z 1005.825,A -85,B 0,C 180,E1 7437.786,E2 7437.786} C_VEL
LIN {X 0,Y 619.57,Z 1074.847,A -85,B 0,C 180,E1 7439.552,E2 7439.552} C_VEL
LIN {X 0,Y 614.349,Z 1141.966,A -85,B 0,C 180,E1 7442.778,E2 7442.778} C_VEL
LIN {X 0,Y 609.386,Z 1200.193,A -85,B 0,C 180,E1 7447.218,E2 7447.218} C_VEL
LIN {X 0,Y 605.833,Z 1245.168,A -85,B 0,C 180,E1 7452.423,E2 7452.423} C_VEL
LIN {X 0,Y 603.779,Z 1275.64,A -85,B 0,C 180,E1 7458.013,E2 7458.013} C_VEL
LIN {X 0,Y 603,Z 1293.346,A -85,B 0,C 180,E1 7463.722,E2 7463.722} C_VEL
LIN {X 0,Y 602.898,Z 1299.822,A -85,B 0,C 180,E1 7469.315,E2 7469.315} C_VEL
LIN {X 0,Y 603.049,Z 1295.695,A -85,B 0,C 180,E1 7475.088,E2 7475.088} C_VEL
LIN {X 0,Y 603.996,Z 1277.931,A -85,B 0,C 180,E1 7481.397,E2 7481.397} C_VEL
LIN {X 0,Y 606.04,Z 1247.08,A -85,B 0,C 180,E1 7487.293,E2 7487.293} C_VEL
LIN {X 0,Y 609.012,Z 1202.729,A -85,B 0,C 180,E1 7492.271,E2 7492.271} C_VEL
LIN {X 0,Y 612.488,Z 1146.505,A -85,B 0,C 180,E1 7496.299,E2 7496.299} C_VEL
LIN {X 0,Y 615.915,Z 1076.981,A -85,B 0,C 180,E1 7499.424,E2 7499.424} C_VEL
LIN {X 0,Y 617.847,Z 996.189,A -85,B 0,C 180,E1 7501.413,E2 7501.413} C_VEL
LIN {X 0,Y 604.874,Z 958.099,A -85,B 0,C 180,E1 7502.415,E2 7502.415} C_VEL
LIN {X 0,Y 602.302,Z 948.94,A -85,B 0,C 180,E1 7502.836,E2 7502.836} C_VEL
LIN {X 0,Y 602.043,Z 948.94,A -85,B 0,C 180,E1 7511.972,E2 7511.972} C_VEL
LIN {X 0,Y 601.954,Z 948.94,A -85,B 0,C 180,E1 7520.3,E2 7520.3} C_VEL
LIN {X 0,Y 602.494,Z 950.806,A -85,B 0,C 180,E1 7524.992,E2 7524.992} C_VEL
LIN {X 0,Y 618.32,Z 1002.184,A -85,B 0,C 180,E1 7526.68,E2 7526.68} C_VEL
LIN {X 0,Y 615.17,Z 1065.212,A -85,B 0,C 180,E1 7529.249,E2 7529.249} C_VEL
LIN {X 0,Y 611.034,Z 1119.915,A -85,B 0,C 180,E1 7533.026,E2 7533.026} C_VEL
LIN {X 0,Y 607.027,Z 1166.152,A -85,B 0,C 180,E1 7538.027,E2 7538.027} C_VEL
LIN {X 0,Y 604.445,Z 1201.152,A -85,B 0,C 180,E1 7543.98,E2 7543.98} C_VEL
LIN {X 0,Y 603.45,Z 1221.624,A -85,B 0,C 180,E1 7549.874,E2 7549.874} C_VEL
LIN {X 0,Y 603.173,Z 1229.285,A -85,B 0,C 180,E1 7554.961,E2 7554.961} C_VEL
LIN {X 0,Y 603.22,Z 1227.627,A -85,B 0,C 180,E1 7560.735,E2 7560.735} C_VEL
LIN {X 0,Y 603.56,Z 1213.339,A -85,B 0,C 180,E1 7566.875,E2 7566.875} C_VEL
LIN {X 0,Y 604.946,Z 1185.959,A -85,B 0,C 180,E1 7572.881,E2 7572.881} C_VEL
LIN {X 0,Y 608.399,Z 1146.119,A -85,B 0,C 180,E1 7578.367,E2 7578.367} C_VEL
LIN {X 0,Y 613.482,Z 1093.229,A -85,B 0,C 180,E1 7583.069,E2 7583.069} C_VEL
LIN {X 0,Y 618.396,Z 1032.11,A -85,B 0,C 180,E1 7586.485,E2 7586.485} C_VEL
LIN {X 0,Y 618.784,Z 991.312,A -85,B 0,C 180,E1 7588.021,E2 7588.021} C_VEL
LIN {X 0,Y 602.285,Z 948.94,A -85,B 0,C 180,E1 7590.074,E2 7590.074} C_VEL
LIN {X 0,Y 601.991,Z 948.94,A -85,B 0,C 180,E1 7598.168,E2 7598.168} C_VEL
LIN {X 0,Y 602.103,Z 948.94,A -85,B 0,C 180,E1 7606.084,E2 7606.084} C_VEL
LIN {X 0,Y 602.113,Z 948.94,A -85,B 0,C 180,E1 7615.035,E2 7615.035} C_VEL
LIN {X 0,Y 602.219,Z 948.94,A -85,B 0,C 180,E1 7623.799,E2 7623.799} C_VEL
LIN {X 0,Y 602.623,Z 950.198,A -85,B 0,C 180,E1 7631.134,E2 7631.134} C_VEL
LIN {X 0,Y 609.485,Z 982.889,A -85,B 0,C 180,E1 7631.752,E2 7631.752} C_VEL
LIN {X 0,Y 609.162,Z 1040.383,A -85,B 0,C 180,E1 7632.906,E2 7632.906} C_VEL
LIN {X 0,Y 607.396,Z 1086.061,A -85,B 0,C 180,E1 7635.313,E2 7635.313} C_VEL
LIN {X 0,Y 605.388,Z 1122.804,A -85,B 0,C 180,E1 7638.951,E2 7638.951} C_VEL
LIN {X 0,Y 604.058,Z 1146.706,A -85,B 0,C 180,E1 7643.474,E2 7643.474} C_VEL
LIN {X 0,Y 603.682,Z 1155.56,A -85,B 0,C 180,E1 7647.804,E2 7647.804} C_VEL
LIN {X 0,Y 603.802,Z 1152.917,A -85,B 0,C 180,E1 7652.125,E2 7652.125} C_VEL
LIN {X 0,Y 604.467,Z 1136.817,A -85,B 0,C 180,E1 7656.716,E2 7656.716} C_VEL
LIN {X 0,Y 606.092,Z 1107.084,A -85,B 0,C 180,E1 7660.786,E2 7660.786} C_VEL
LIN {X 0,Y 608.13,Z 1066.01,A -85,B 0,C 180,E1 7663.859,E2 7663.859} C_VEL
LIN {X 0,Y 609.653,Z 1017.981,A -85,B 0,C 180,E1 7665.628,E2 7665.628} C_VEL
LIN {X 0,Y 607.24,Z 966.591,A -85,B 0,C 180,E1 7666.411,E2 7666.411} C_VEL
LIN {X 0,Y 602.479,Z 948.94,A -85,B 0,C 180,E1 7666.798,E2 7666.798} C_VEL
LIN {X 0,Y 601.915,Z 948.94,A -85,B 0,C 180,E1 7674.538,E2 7674.538} C_VEL
LIN {X 0,Y 601.934,Z 948.94,A -85,B 0,C 180,E1 7682.773,E2 7682.773} C_VEL
LIN {X 0,Y 601.921,Z 948.94,A -85,B 0,C 180,E1 7689.953,E2 7689.953} C_VEL
LIN {X 0,Y 602.097,Z 948.94,A -85,B 0,C 180,E1 7698.066,E2 7698.066} C_VEL
LIN {X 0,Y 602.16,Z 948.94,A -85,B 0,C 180,E1 7707.168,E2 7707.168} C_VEL
LIN {X 0,Y 602.353,Z 948.94,A -85,B 0,C 180,E1 7715.417,E2 7715.417} C_VEL
LIN {X 0,Y 602.853,Z 948.94,A -85,B 0,C 180,E1 7724.657,E2 7724.657} C_VEL
LIN {X 0,Y 602.512,Z 948.94,A -85,B 0,C 180,E1 7732.022,E2 7732.022} C_VEL
LIN {X 0,Y 602.627,Z 948.94,A -85,B 0,C 180,E1 7739.264,E2 7739.264} C_VEL
LIN {X 0,Y 602.718,Z 948.94,A -85,B 0,C 180,E1 7746.493,E2 7746.493} C_VEL
LIN {X 0,Y 602.277,Z 948.94,A -85,B 0,C 180,E1 7755.329,E2 7755.329} C_VEL
LIN {X 0,Y 602.085,Z 948.94,A -85,B 0,C 180,E1 7763.193,E2 7763.193} C_VEL
LIN {X 0,Y 602.48,Z 948.94,A -85,B 0,C 180,E1 7771.078,E2 7771.078} C_VEL
LIN {X 0,Y 602.312,Z 948.94,A -85,B 0,C 180,E1 7779.967,E2 7779.967} C_VEL
LIN {X 0,Y 602.15,Z 948.94,A -85,B 0,C 180,E1 7788.156,E2 7788.156} C_VEL
LIN {X 0,Y 602.479,Z 948.94,A -85,B 0,C 180,E1 7793.992,E2 7793.992} C_VEL
LIN {X 0,Y 598.906,Z 958.403,A -85,B 0,C 180,E1 7795.264,E2 7795.264} C_VEL
LIN {X 0,Y 599.459,Z 965.322,A -85,B 0,C 180,E1 7795.639,E2 7795.639} C_VEL
LIN {X 0,Y 616.556,Z 1008.045,A -85,B 0,C 180,E1 7797.429,E2 7797.429} C_VEL
LIN {X 0,Y 612.223,Z 1077.704,A -85,B 0,C 180,E1 7799.317,E2 7799.317} C_VEL
LIN {X 0,Y 606.638,Z 1144.774,A -85,B 0,C 180,E1 7802.672,E2 7802.672} C_VEL
LIN {X 0,Y 601.408,Z 1202.859,A -85,B 0,C 180,E1 7807.265,E2 7807.265} C_VEL
LIN {X 0,Y 597.787,Z 1246.98,A -85,B 0,C 180,E1 7812.574,E2 7812.574} C_VEL
LIN {X 0,Y 595.782,Z 1276.946,A -85,B 0,C 180,E1 7818.191,E2 7818.191} C_VEL
LIN {X 0,Y 595.017,Z 1292.959,A -85,B 0,C 180,E1 7823.447,E2 7823.447} C_VEL
LIN {X 0,Y 595.087,Z 1299.183,A -85,B 0,C 180,E1 7827.844,E2 7827.844} C_VEL
LIN {X 0,Y 594.967,Z 1297.762,A -85,B 0,C 180,E1 7833.691,E2 7833.691} C_VEL
LIN {X 0,Y 595.313,Z 1284.923,A -85,B 0,C 180,E1 7839.572,E2 7839.572} C_VEL
LIN {X 0,Y 596.569,Z 1261.81,A -85,B 0,C 180,E1 7844.969,E2 7844.969} C_VEL
LIN {X 0,Y 599.16,Z 1225.349,A -85,B 0,C 180,E1 7850.029,E2 7850.029} C_VEL
LIN {X 0,Y 602.734,Z 1176.041,A -85,B 0,C 180,E1 7854.482,E2 7854.482} C_VEL
LIN {X 0,Y 606.52,Z 1111.157,A -85,B 0,C 180,E1 7858.216,E2 7858.216} C_VEL
LIN {X 0,Y 609.972,Z 1034.71,A -85,B 0,C 180,E1 7860.839,E2 7860.839} C_VEL
LIN {X 0,Y 609.145,Z 996.272,A -85,B 0,C 180,E1 7861.698,E2 7861.698} C_VEL
LIN {X 0,Y 594.226,Z 948.94,A -85,B 0,C 180,E1 7863.129,E2 7863.129} C_VEL
LIN {X 0,Y 594.016,Z 948.94,A -85,B 0,C 180,E1 7872.649,E2 7872.649} C_VEL
LIN {X 0,Y 593.963,Z 948.94,A -85,B 0,C 180,E1 7881.258,E2 7881.258} C_VEL
LIN {X 0,Y 594.367,Z 950.362,A -85,B 0,C 180,E1 7884.644,E2 7884.644} C_VEL
LIN {X 0,Y 610.928,Z 1004.589,A -85,B 0,C 180,E1 7886.451,E2 7886.451} C_VEL
LIN {X 0,Y 607.647,Z 1066.953,A -85,B 0,C 180,E1 7889.039,E2 7889.039} C_VEL
LIN {X 0,Y 603.459,Z 1120.512,A -85,B 0,C 180,E1 7892.779,E2 7892.779} C_VEL
LIN {X 0,Y 599.247,Z 1167.099,A -85,B 0,C 180,E1 7897.869,E2 7897.869} C_VEL
LIN {X 0,Y 596.578,Z 1201.052,A -85,B 0,C 180,E1 7903.763,E2 7903.763} C_VEL
LIN {X 0,Y 595.513,Z 1221.514,A -85,B 0,C 180,E1 7909.737,E2 7909.737} C_VEL
LIN {X 0,Y 595.181,Z 1229.246,A -85,B 0,C 180,E1 7914.894,E2 7914.894} C_VEL
LIN {X 0,Y 595.23,Z 1227.679,A -85,B 0,C 180,E1 7920.745,E2 7920.745} C_VEL
LIN {X 0,Y 595.565,Z 1213.472,A -85,B 0,C 180,E1 7926.967,E2 7926.967} C_VEL
LIN {X 0,Y 597.124,Z 1186.526,A -85,B 0,C 180,E1 7933.052,E2 7933.052} C_VEL
LIN {X 0,Y 600.783,Z 1146.631,A -85,B 0,C 180,E1 7938.616,E2 7938.616} C_VEL
LIN {X 0,Y 606.164,Z 1093.232,A -85,B 0,C 180,E1 7943.411,E2 7943.411} C_VEL
LIN {X 0,Y 611.374,Z 1031.233,A -85,B 0,C 180,E1 7946.884,E2 7946.884} C_VEL
LIN {X 0,Y 611.506,Z 993.286,A -85,B 0,C 180,E1 7948.343,E2 7948.343} C_VEL
LIN {X 0,Y 594.174,Z 948.94,A -85,B 0,C 180,E1 7950.518,E2 7950.518} C_VEL
LIN {X 0,Y 593.917,Z 948.94,A -85,B 0,C 180,E1 7958.783,E2 7958.783} C_VEL
LIN {X 0,Y 593.995,Z 948.94,A -85,B 0,C 180,E1 7967.349,E2 7967.349} C_VEL
LIN {X 0,Y 594.062,Z 948.94,A -85,B 0,C 180,E1 7976.162,E2 7976.162} C_VEL
LIN {X 0,Y 594.278,Z 948.94,A -85,B 0,C 180,E1 7985.085,E2 7985.085} C_VEL
LIN {X 0,Y 594.727,Z 950.682,A -85,B 0,C 180,E1 7990.88,E2 7990.88} C_VEL
LIN {X 0,Y 601.925,Z 984.602,A -85,B 0,C 180,E1 7991.536,E2 7991.536} C_VEL
LIN {X 0,Y 601.554,Z 1040.79,A -85,B 0,C 180,E1 7992.676,E2 7992.676} C_VEL
LIN {X 0,Y 599.801,Z 1085.636,A -85,B 0,C 180,E1 7995.029,E2 7995.029} C_VEL
LIN {X 0,Y 597.858,Z 1121.34,A -85,B 0,C 180,E1 7998.505,E2 7998.505} C_VEL
LIN {X 0,Y 596.567,Z 1145.049,A -85,B 0,C 180,E1 8002.7,E2 8002.7} C_VEL
LIN {X 0,Y 596.112,Z 1154.831,A -85,B 0,C 180,E1 8006.316,E2 8006.316} C_VEL
LIN {X 0,Y 596.038,Z 1155.09,A -85,B 0,C 180,E1 8011.423,E2 8011.423} C_VEL
LIN {X 0,Y 596.552,Z 1140.922,A -85,B 0,C 180,E1 8016.169,E2 8016.169} C_VEL
LIN {X 0,Y 598.117,Z 1113.241,A -85,B 0,C 180,E1 8020.377,E2 8020.377} C_VEL
LIN {X 0,Y 600.271,Z 1073.956,A -85,B 0,C 180,E1 8023.64,E2 8023.64} C_VEL
LIN {X 0,Y 601.822,Z 1026.88,A -85,B 0,C 180,E1 8025.649,E2 8025.649} C_VEL
LIN {X 0,Y 599.958,Z 969.208,A -85,B 0,C 180,E1 8026.604,E2 8026.604} C_VEL
LIN {X 0,Y 594.454,Z 948.94,A -85,B 0,C 180,E1 8027.031,E2 8027.031} C_VEL
LIN {X 0,Y 593.906,Z 948.94,A -85,B 0,C 180,E1 8034.891,E2 8034.891} C_VEL
LIN {X 0,Y 593.88,Z 948.94,A -85,B 0,C 180,E1 8043.812,E2 8043.812} C_VEL
LIN {X 0,Y 593.988,Z 948.94,A -85,B 0,C 180,E1 8053.239,E2 8053.239} C_VEL
LIN {X 0,Y 594.117,Z 948.94,A -85,B 0,C 180,E1 8061.233,E2 8061.233} C_VEL
LIN {X 0,Y 594.305,Z 948.94,A -85,B 0,C 180,E1 8070.115,E2 8070.115} C_VEL
LIN {X 0,Y 594.484,Z 948.94,A -85,B 0,C 180,E1 8078.582,E2 8078.582} C_VEL
LIN {X 0,Y 595.239,Z 948.94,A -85,B 0,C 180,E1 8087.468,E2 8087.468} C_VEL
LIN {X 0,Y 595.242,Z 948.94,A -85,B 0,C 180,E1 8097.794,E2 8097.794} C_VEL
LIN {X 0,Y 594.685,Z 948.94,A -85,B 0,C 180,E1 8106.581,E2 8106.581} C_VEL
LIN {X 0,Y 594.232,Z 948.94,A -85,B 0,C 180,E1 8115.542,E2 8115.542} C_VEL
LIN {X 0,Y 594.065,Z 948.94,A -85,B 0,C 180,E1 8123.314,E2 8123.314} C_VEL
LIN {X 0,Y 594.439,Z 948.94,A -85,B 0,C 180,E1 8131.546,E2 8131.546} C_VEL
LIN {X 0,Y 594.227,Z 948.94,A -85,B 0,C 180,E1 8140.623,E2 8140.623} C_VEL
LIN {X 0,Y 594.207,Z 948.94,A -85,B 0,C 180,E1 8149.421,E2 8149.421} C_VEL
LIN {X 0,Y 594.573,Z 949.573,A -85,B 0,C 180,E1 8154.437,E2 8154.437} C_VEL
LIN {X 0,Y 599.459,Z 965.322,A -85,B 0,C 180,E1 8155.639,E2 8155.639} C_VEL
LIN {X 0,Y 605.028,Z 998.92,A -85,B 0,C 180,E1 8156.568,E2 8156.568} C_VEL
LIN {X 0,Y 609.572,Z 1012.235,A -85,B 0,C 180,E1 8157.104,E2 8157.104} C_VEL
LIN {X 0,Y 604.666,Z 1083.061,A -85,B 0,C 180,E1 8159.183,E2 8159.183} C_VEL
LIN {X 0,Y 598.782,Z 1148.183,A -85,B 0,C 180,E1 8162.61,E2 8162.61} C_VEL
LIN {X 0,Y 593.403,Z 1205.702,A -85,B 0,C 180,E1 8167.351,E2 8167.351} C_VEL
LIN {X 0,Y 589.691,Z 1249.436,A -85,B 0,C 180,E1 8172.827,E2 8172.827} C_VEL
LIN {X 0,Y 587.753,Z 1279.794,A -85,B 0,C 180,E1 8178.874,E2 8178.874} C_VEL
LIN {X 0,Y 587.23,Z 1295.785,A -85,B 0,C 180,E1 8184.848,E2 8184.848} C_VEL
LIN {X 0,Y 587.486,Z 1299.8,A -85,B 0,C 180,E1 8190.776,E2 8190.776} C_VEL
LIN {X 0,Y 587.584,Z 1291.122,A -85,B 0,C 180,E1 8197.455,E2 8197.455} C_VEL
LIN {X 0,Y 588.432,Z 1269.566,A -85,B 0,C 180,E1 8203.456,E2 8203.456} C_VEL
LIN {X 0,Y 590.764,Z 1234.487,A -85,B 0,C 180,E1 8208.958,E2 8208.958} C_VEL
LIN {X 0,Y 594.174,Z 1186.369,A -85,B 0,C 180,E1 8213.754,E2 8213.754} C_VEL
LIN {X 0,Y 598.029,Z 1123.268,A -85,B 0,C 180,E1 8217.768,E2 8217.768} C_VEL
LIN {X 0,Y 601.676,Z 1047.886,A -85,B 0,C 180,E1 8220.696,E2 8220.696} C_VEL
LIN {X 0,Y 601.555,Z 998.382,A -85,B 0,C 180,E1 8221.914,E2 8221.914} C_VEL
LIN {X 0,Y 586.145,Z 948.94,A -85,B 0,C 180,E1 8223.571,E2 8223.571} C_VEL
LIN {X 0,Y 586.012,Z 948.94,A -85,B 0,C 180,E1 8232.446,E2 8232.446} C_VEL
LIN {X 0,Y 585.885,Z 948.94,A -85,B 0,C 180,E1 8240.621,E2 8240.621} C_VEL
LIN {X 0,Y 586.486,Z 950.938,A -85,B 0,C 180,E1 8244.3,E2 8244.3} C_VEL
LIN {X 0,Y 603.572,Z 1006.204,A -85,B 0,C 180,E1 8246.188,E2 8246.188} C_VEL
LIN {X 0,Y 600.195,Z 1068.159,A -85,B 0,C 180,E1 8248.791,E2 8248.791} C_VEL
LIN {X 0,Y 595.754,Z 1122.415,A -85,B 0,C 180,E1 8252.643,E2 8252.643} C_VEL
LIN {X 0,Y 591.452,Z 1168.627,A -85,B 0,C 180,E1 8257.787,E2 8257.787} C_VEL
LIN {X 0,Y 588.539,Z 1202.951,A -85,B 0,C 180,E1 8263.92,E2 8263.92} C_VEL
LIN {X 0,Y 587.269,Z 1223.002,A -85,B 0,C 180,E1 8270.344,E2 8270.344} C_VEL
LIN {X 0,Y 586.901,Z 1229.818,A -85,B 0,C 180,E1 8276.308,E2 8276.308} C_VEL
LIN {X 0,Y 586.945,Z 1225.542,A -85,B 0,C 180,E1 8282.238,E2 8282.238} C_VEL
LIN {X 0,Y 587.941,Z 1208.685,A -85,B 0,C 180,E1 8288.551,E2 8288.551} C_VEL
LIN {X 0,Y 590.424,Z 1177.148,A -85,B 0,C 180,E1 8294.874,E2 8294.874} C_VEL
LIN {X 0,Y 594.822,Z 1133.019,A -85,B 0,C 180,E1 8300.36,E2 8300.36} C_VEL
LIN {X 0,Y 600.324,Z 1078.207,A -85,B 0,C 180,E1 8304.771,E2 8304.771} C_VEL
LIN {X 0,Y 605.379,Z 1015.677,A -85,B 0,C 180,E1 8307.875,E2 8307.875} C_VEL
LIN {X 0,Y 603.889,Z 994.124,A -85,B 0,C 180,E1 8308.727,E2 8308.727} C_VEL
LIN {X 0,Y 586.081,Z 948.94,A -85,B 0,C 180,E1 8310.906,E2 8310.906} C_VEL
LIN {X 0,Y 585.772,Z 948.94,A -85,B 0,C 180,E1 8320.116,E2 8320.116} C_VEL
LIN {X 0,Y 585.972,Z 948.94,A -85,B 0,C 180,E1 8328.63,E2 8328.63} C_VEL
LIN {X 0,Y 586.089,Z 948.94,A -85,B 0,C 180,E1 8337.904,E2 8337.904} C_VEL
LIN {X 0,Y 586.46,Z 948.94,A -85,B 0,C 180,E1 8346.783,E2 8346.783} C_VEL
LIN {X 0,Y 586.65,Z 950.49,A -85,B 0,C 180,E1 8350.604,E2 8350.604} C_VEL
LIN {X 0,Y 594.366,Z 985.609,A -85,B 0,C 180,E1 8351.306,E2 8351.306} C_VEL
LIN {X 0,Y 593.946,Z 1042.22,A -85,B 0,C 180,E1 8352.476,E2 8352.476} C_VEL
LIN {X 0,Y 592.028,Z 1087.664,A -85,B 0,C 180,E1 8354.923,E2 8354.923} C_VEL
LIN {X 0,Y 589.883,Z 1123.885,A -85,B 0,C 180,E1 8358.57,E2 8358.57} C_VEL
LIN {X 0,Y 588.487,Z 1147.228,A -85,B 0,C 180,E1 8362.929,E2 8362.929} C_VEL
LIN {X 0,Y 587.828,Z 1157.447,A -85,B 0,C 180,E1 8367.745,E2 8367.745} C_VEL
LIN {X 0,Y 587.96,Z 1154.864,A -85,B 0,C 180,E1 8372.182,E2 8372.182} C_VEL
LIN {X 0,Y 588.725,Z 1138.979,A -85,B 0,C 180,E1 8376.866,E2 8376.866} C_VEL
LIN {X 0,Y 590.533,Z 1109.182,A -85,B 0,C 180,E1 8381.073,E2 8381.073} C_VEL
LIN {X 0,Y 592.796,Z 1068.232,A -85,B 0,C 180,E1 8384.224,E2 8384.224} C_VEL
LIN {X 0,Y 594.422,Z 1019.896,A -85,B 0,C 180,E1 8386.057,E2 8386.057} C_VEL
LIN {X 0,Y 592.018,Z 969.351,A -85,B 0,C 180,E1 8386.853,E2 8386.853} C_VEL
LIN {X 0,Y 586.445,Z 948.94,A -85,B 0,C 180,E1 8387.465,E2 8387.465} C_VEL
LIN {X 0,Y 586.077,Z 948.94,A -85,B 0,C 180,E1 8396.898,E2 8396.898} C_VEL
LIN {X 0,Y 585.973,Z 948.94,A -85,B 0,C 180,E1 8405.588,E2 8405.588} C_VEL
LIN {X 0,Y 586.118,Z 948.94,A -85,B 0,C 180,E1 8415.336,E2 8415.336} C_VEL
LIN {X 0,Y 586.125,Z 948.94,A -85,B 0,C 180,E1 8424.566,E2 8424.566} C_VEL
LIN {X 0,Y 586.186,Z 948.94,A -85,B 0,C 180,E1 8433.17,E2 8433.17} C_VEL
LIN {X 0,Y 586.308,Z 948.94,A -85,B 0,C 180,E1 8441.104,E2 8441.104} C_VEL
LIN {X 0,Y 587.241,Z 948.94,A -85,B 0,C 180,E1 8448.808,E2 8448.808} C_VEL
LIN {X 0,Y 587.236,Z 948.94,A -85,B 0,C 180,E1 8457.764,E2 8457.764} C_VEL
LIN {X 0,Y 586.652,Z 948.94,A -85,B 0,C 180,E1 8466.671,E2 8466.671} C_VEL
LIN {X 0,Y 586.521,Z 948.94,A -85,B 0,C 180,E1 8474.217,E2 8474.217} C_VEL
LIN {X 0,Y 586.066,Z 948.94,A -85,B 0,C 180,E1 8483.304,E2 8483.304} C_VEL
LIN {X 0,Y 586.379,Z 948.94,A -85,B 0,C 180,E1 8492.031,E2 8492.031} C_VEL
LIN {X 0,Y 586.229,Z 948.94,A -85,B 0,C 180,E1 8501.297,E2 8501.297} C_VEL
LIN {X 0,Y 586.261,Z 948.94,A -85,B 0,C 180,E1 8510.696,E2 8510.696} C_VEL
LIN {X 0,Y 586.644,Z 950.492,A -85,B 0,C 180,E1 8514.086,E2 8514.086} C_VEL
LIN {X 0,Y 592.886,Z 968.096,A -85,B 0,C 180,E1 8515.25,E2 8515.25} C_VEL
LIN {X 0,Y 605.028,Z 998.92,A -85,B 0,C 180,E1 8516.568,E2 8516.568} C_VEL
LIN {X 0,Y 602.242,Z 1022.472,A -85,B 0,C 180,E1 8516.917,E2 8516.917} C_VEL
LIN {X 0,Y 596.667,Z 1091.878,A -85,B 0,C 180,E1 8519.208,E2 8519.208} C_VEL
LIN {X 0,Y 590.508,Z 1156.588,A -85,B 0,C 180,E1 8522.91,E2 8522.91} C_VEL
LIN {X 0,Y 585.075,Z 1211.857,A -85,B 0,C 180,E1 8527.809,E2 8527.809} C_VEL
LIN {X 0,Y 581.5,Z 1254.43,A -85,B 0,C 180,E1 8533.554,E2 8533.554} C_VEL
LIN {X 0,Y 579.884,Z 1283.44,A -85,B 0,C 180,E1 8539.922,E2 8539.922} C_VEL
LIN {X 0,Y 579.54,Z 1297.711,A -85,B 0,C 180,E1 8546.284,E2 8546.284} C_VEL
LIN {X 0,Y 579.364,Z 1298.974,A -85,B 0,C 180,E1 8552.288,E2 8552.288} C_VEL
LIN {X 0,Y 579.372,Z 1287.586,A -85,B 0,C 180,E1 8558.698,E2 8558.698} C_VEL
LIN {X 0,Y 580.489,Z 1264.304,A -85,B 0,C 180,E1 8564.416,E2 8564.416} C_VEL
LIN {X 0,Y 583.057,Z 1227.726,A -85,B 0,C 180,E1 8569.812,E2 8569.812} C_VEL
LIN {X 0,Y 586.787,Z 1176.593,A -85,B 0,C 180,E1 8574.58,E2 8574.58} C_VEL
LIN {X 0,Y 590.787,Z 1111.372,A -85,B 0,C 180,E1 8578.481,E2 8578.481} C_VEL
LIN {X 0,Y 594.683,Z 1033.408,A -85,B 0,C 180,E1 8581.308,E2 8581.308} C_VEL
LIN {X 0,Y 593.948,Z 1000.496,A -85,B 0,C 180,E1 8582.143,E2 8582.143} C_VEL
LIN {X 0,Y 578.128,Z 948.94,A -85,B 0,C 180,E1 8583.848,E2 8583.848} C_VEL
LIN {X 0,Y 577.993,Z 948.94,A -85,B 0,C 180,E1 8592.07,E2 8592.07} C_VEL
LIN {X 0,Y 577.873,Z 948.94,A -85,B 0,C 180,E1 8600.823,E2 8600.823} C_VEL
LIN {X 0,Y 578.395,Z 950.667,A -85,B 0,C 180,E1 8603.913,E2 8603.913} C_VEL
LIN {X 0,Y 596.235,Z 1009.366,A -85,B 0,C 180,E1 8605.959,E2 8605.959} C_VEL
LIN {X 0,Y 592.686,Z 1071.134,A -85,B 0,C 180,E1 8608.631,E2 8608.631} C_VEL
LIN {X 0,Y 587.897,Z 1125.794,A -85,B 0,C 180,E1 8612.638,E2 8612.638} C_VEL
LIN {X 0,Y 583.629,Z 1170.02,A -85,B 0,C 180,E1 8617.694,E2 8617.694} C_VEL
LIN {X 0,Y 580.743,Z 1203.181,A -85,B 0,C 180,E1 8623.698,E2 8623.698} C_VEL
LIN {X 0,Y 579.333,Z 1223.386,A -85,B 0,C 180,E1 8630.21,E2 8630.21} C_VEL
LIN {X 0,Y 578.939,Z 1230.058,A -85,B 0,C 180,E1 8636.257,E2 8636.257} C_VEL
LIN {X 0,Y 578.964,Z 1225.986,A -85,B 0,C 180,E1 8642.268,E2 8642.268} C_VEL
LIN {X 0,Y 579.875,Z 1210.663,A -85,B 0,C 180,E1 8648.292,E2 8648.292} C_VEL
LIN {X 0,Y 582.065,Z 1182.158,A -85,B 0,C 180,E1 8654.358,E2 8654.358} C_VEL
LIN {X 0,Y 586.618,Z 1139.164,A -85,B 0,C 180,E1 8660.065,E2 8660.065} C_VEL
LIN {X 0,Y 592.48,Z 1084.62,A -85,B 0,C 180,E1 8664.711,E2 8664.711} C_VEL
LIN {X 0,Y 597.812,Z 1023.056,A -85,B 0,C 180,E1 8667.965,E2 8667.965} C_VEL
LIN {X 0,Y 597.265,Z 997.769,A -85,B 0,C 180,E1 8668.971,E2 8668.971} C_VEL
LIN {X 0,Y 578.009,Z 948.94,A -85,B 0,C 180,E1 8671.376,E2 8671.376} C_VEL
LIN {X 0,Y 577.786,Z 948.94,A -85,B 0,C 180,E1 8680.08,E2 8680.08} C_VEL
LIN {X 0,Y 577.96,Z 948.94,A -85,B 0,C 180,E1 8688.478,E2 8688.478} C_VEL
LIN {X 0,Y 578.08,Z 948.94,A -85,B 0,C 180,E1 8697.405,E2 8697.405} C_VEL
LIN {X 0,Y 578.305,Z 948.94,A -85,B 0,C 180,E1 8705.964,E2 8705.964} C_VEL
LIN {X 0,Y 578.513,Z 948.94,A -85,B 0,C 180,E1 8710.292,E2 8710.292} C_VEL
LIN {X 0,Y 586.801,Z 986.384,A -85,B 0,C 180,E1 8711.065,E2 8711.065} C_VEL
LIN {X 0,Y 586.374,Z 1042.482,A -85,B 0,C 180,E1 8712.229,E2 8712.229} C_VEL
LIN {X 0,Y 584.433,Z 1087.248,A -85,B 0,C 180,E1 8714.626,E2 8714.626} C_VEL
LIN {X 0,Y 582.273,Z 1123.125,A -85,B 0,C 180,E1 8718.199,E2 8718.199} C_VEL
LIN {X 0,Y 580.819,Z 1146.698,A -85,B 0,C 180,E1 8722.458,E2 8722.458} C_VEL
LIN {X 0,Y 580.244,Z 1156.704,A -85,B 0,C 180,E1 8726.215,E2 8726.215} C_VEL
LIN {X 0,Y 580.186,Z 1157.025,A -85,B 0,C 180,E1 8731.462,E2 8731.462} C_VEL
LIN {X 0,Y 580.774,Z 1143.051,A -85,B 0,C 180,E1 8736.307,E2 8736.307} C_VEL
LIN {X 0,Y 582.514,Z 1115.319,A -85,B 0,C 180,E1 8740.658,E2 8740.658} C_VEL
LIN {X 0,Y 584.946,Z 1075.657,A -85,B 0,C 180,E1 8744.036,E2 8744.036} C_VEL
LIN {X 0,Y 586.558,Z 1028.525,A -85,B 0,C 180,E1 8746.092,E2 8746.092} C_VEL
LIN {X 0,Y 584.925,Z 972.619,A -85,B 0,C 180,E1 8747.041,E2 8747.041} C_VEL
LIN {X 0,Y 578.448,Z 948.94,A -85,B 0,C 180,E1 8747.715,E2 8747.715} C_VEL
LIN {X 0,Y 578.042,Z 948.94,A -85,B 0,C 180,E1 8757.303,E2 8757.303} C_VEL
LIN {X 0,Y 577.887,Z 948.94,A -85,B 0,C 180,E1 8766.743,E2 8766.743} C_VEL
LIN {X 0,Y 578.104,Z 948.94,A -85,B 0,C 180,E1 8776.146,E2 8776.146} C_VEL
LIN {X 0,Y 578.073,Z 948.94,A -85,B 0,C 180,E1 8785.703,E2 8785.703} C_VEL
LIN {X 0,Y 578.257,Z 948.94,A -85,B 0,C 180,E1 8794.767,E2 8794.767} C_VEL
LIN {X 0,Y 578.644,Z 948.94,A -85,B 0,C 180,E1 8803.998,E2 8803.998} C_VEL
LIN {X 0,Y 578.58,Z 948.94,A -85,B 0,C 180,E1 8811.689,E2 8811.689} C_VEL
LIN {X 0,Y 578.651,Z 948.94,A -85,B 0,C 180,E1 8819.234,E2 8819.234} C_VEL
LIN {X 0,Y 578.621,Z 948.94,A -85,B 0,C 180,E1 8826.764,E2 8826.764} C_VEL
LIN {X 0,Y 578.452,Z 948.94,A -85,B 0,C 180,E1 8834.419,E2 8834.419} C_VEL
LIN {X 0,Y 578.148,Z 948.94,A -85,B 0,C 180,E1 8842.359,E2 8842.359} C_VEL
LIN {X 0,Y 578.34,Z 948.94,A -85,B 0,C 180,E1 8851.572,E2 8851.572} C_VEL
LIN {X 0,Y 578.204,Z 948.94,A -85,B 0,C 180,E1 8860.007,E2 8860.007} C_VEL
LIN {X 0,Y 578.224,Z 948.94,A -85,B 0,C 180,E1 8870.041,E2 8870.041} C_VEL
LIN {X 0,Y 578.745,Z 950.919,A -85,B 0,C 180,E1 8873.693,E2 8873.693} C_VEL
LIN {X 0,Y 592.399,Z 986.093,A -85,B 0,C 180,E1 8875.531,E2 8875.531} C_VEL
LIN {X 0,Y 602.659,Z 1014.292,A -85,B 0,C 180,E1 8876.746,E2 8876.746} C_VEL
LIN {X 0,Y 602.242,Z 1022.472,A -85,B 0,C 180,E1 8876.917,E2 8876.917} C_VEL
LIN {X 0,Y 592.566,Z 1056.156,A -85,B 0,C 180,E1 8877.446,E2 8877.446} C_VEL
LIN {X 0,Y 585.91,Z 1126.681,A -85,B 0,C 180,E1 8880.657,E2 8880.657} C_VEL
LIN {X 0,Y 579.734,Z 1187.792,A -85,B 0,C 180,E1 8885.182,E2 8885.182} C_VEL
LIN {X 0,Y 575.008,Z 1237.276,A -85,B 0,C 180,E1 8890.781,E2 8890.781} C_VEL
LIN {X 0,Y 572.312,Z 1270.636,A -85,B 0,C 180,E1 8896.625,E2 8896.625} C_VEL
LIN {X 0,Y 571.285,Z 1290.366,A -85,B 0,C 180,E1 8902.407,E2 8902.407} C_VEL
LIN {X 0,Y 571.128,Z 1298.581,A -85,B 0,C 180,E1 8907.754,E2 8907.754} C_VEL
LIN {X 0,Y 571.002,Z 1296.972,A -85,B 0,C 180,E1 8913.847,E2 8913.847} C_VEL
LIN {X 0,Y 571.381,Z 1284.316,A -85,B 0,C 180,E1 8919.591,E2 8919.591} C_VEL
LIN {X 0,Y 572.667,Z 1260.036,A -85,B 0,C 180,E1 8925.186,E2 8925.186} C_VEL
LIN {X 0,Y 575.482,Z 1221.701,A -85,B 0,C 180,E1 8930.524,E2 8930.524} C_VEL
LIN {X 0,Y 579.322,Z 1169.274,A -85,B 0,C 180,E1 8935.208,E2 8935.208} C_VEL
LIN {X 0,Y 583.459,Z 1102.285,A -85,B 0,C 180,E1 8939.064,E2 8939.064} C_VEL
LIN {X 0,Y 587.703,Z 1022.459,A -85,B 0,C 180,E1 8941.83,E2 8941.83} C_VEL
LIN {X 0,Y 586.117,Z 1002.121,A -85,B 0,C 180,E1 8942.39,E2 8942.39} C_VEL
LIN {X 0,Y 570.076,Z 948.94,A -85,B 0,C 180,E1 8944.294,E2 8944.294} C_VEL
LIN {X 0,Y 569.949,Z 948.94,A -85,B 0,C 180,E1 8952.939,E2 8952.939} C_VEL
LIN {X 0,Y 569.96,Z 948.94,A -85,B 0,C 180,E1 8961.81,E2 8961.81} C_VEL
LIN {X 0,Y 570.259,Z 950.405,A -85,B 0,C 180,E1 8963.499,E2 8963.499} C_VEL
LIN {X 0,Y 588.939,Z 1011.11,A -85,B 0,C 180,E1 8965.676,E2 8965.676} C_VEL
LIN {X 0,Y 585.251,Z 1072.913,A -85,B 0,C 180,E1 8968.393,E2 8968.393} C_VEL
LIN {X 0,Y 580.264,Z 1127.334,A -85,B 0,C 180,E1 8972.458,E2 8972.458} C_VEL
LIN {X 0,Y 575.846,Z 1171.054,A -85,B 0,C 180,E1 8977.547,E2 8977.547} C_VEL
LIN {X 0,Y 572.696,Z 1205.08,A -85,B 0,C 180,E1 8983.858,E2 8983.858} C_VEL
LIN {X 0,Y 571.404,Z 1223.782,A -85,B 0,C 180,E1 8990.073,E2 8990.073} C_VEL
LIN {X 0,Y 570.958,Z 1230.547,A -85,B 0,C 180,E1 8996.204,E2 8996.204} C_VEL
LIN {X 0,Y 570.987,Z 1226.504,A -85,B 0,C 180,E1 9002.3,E2 9002.3} C_VEL
LIN {X 0,Y 571.973,Z 1211.178,A -85,B 0,C 180,E1 9008.407,E2 9008.407} C_VEL
LIN {X 0,Y 574.496,Z 1181.182,A -85,B 0,C 180,E1 9014.801,E2 9014.801} C_VEL
LIN {X 0,Y 579.343,Z 1137.876,A -85,B 0,C 180,E1 9020.528,E2 9020.528} C_VEL
LIN {X 0,Y 585.448,Z 1083.04,A -85,B 0,C 180,E1 9025.188,E2 9025.188} C_VEL
LIN {X 0,Y 591.077,Z 1020.158,A -85,B 0,C 180,E1 9028.463,E2 9028.463} C_VEL
LIN {X 0,Y 589.888,Z 999.283,A -85,B 0,C 180,E1 9029.333,E2 9029.333} C_VEL
LIN {X 0,Y 569.929,Z 948.94,A -85,B 0,C 180,E1 9031.809,E2 9031.809} C_VEL
LIN {X 0,Y 569.755,Z 948.94,A -85,B 0,C 180,E1 9040.763,E2 9040.763} C_VEL
LIN {X 0,Y 569.942,Z 948.94,A -85,B 0,C 180,E1 9049.397,E2 9049.397} C_VEL
LIN {X 0,Y 570.118,Z 948.94,A -85,B 0,C 180,E1 9058.694,E2 9058.694} C_VEL
LIN {X 0,Y 570.386,Z 948.94,A -85,B 0,C 180,E1 9067.271,E2 9067.271} C_VEL
LIN {X 0,Y 570.595,Z 950.191,A -85,B 0,C 180,E1 9070.03,E2 9070.03} C_VEL
LIN {X 0,Y 579.301,Z 989.506,A -85,B 0,C 180,E1 9070.85,E2 9070.85} C_VEL
LIN {X 0,Y 578.754,Z 1045.047,A -85,B 0,C 180,E1 9072.058,E2 9072.058} C_VEL
LIN {X 0,Y 576.566,Z 1090.514,A -85,B 0,C 180,E1 9074.606,E2 9074.606} C_VEL
LIN {X 0,Y 574.227,Z 1126.439,A -85,B 0,C 180,E1 9078.365,E2 9078.365} C_VEL
LIN {X 0,Y 572.496,Z 1150.362,A -85,B 0,C 180,E1 9083.113,E2 9083.113} C_VEL
LIN {X 0,Y 571.975,Z 1159.336,A -85,B 0,C 180,E1 9087.682,E2 9087.682} C_VEL
LIN {X 0,Y 572.1,Z 1156.809,A -85,B 0,C 180,E1 9092.242,E2 9092.242} C_VEL
LIN {X 0,Y 573.03,Z 1140.326,A -85,B 0,C 180,E1 9097.188,E2 9097.188} C_VEL
LIN {X 0,Y 574.987,Z 1111.266,A -85,B 0,C 180,E1 9101.377,E2 9101.377} C_VEL
LIN {X 0,Y 577.476,Z 1070.436,A -85,B 0,C 180,E1 9104.61,E2 9104.61} C_VEL
LIN {X 0,Y 579.19,Z 1021.987,A -85,B 0,C 180,E1 9106.504,E2 9106.504} C_VEL
LIN {X 0,Y 576.993,Z 972.791,A -85,B 0,C 180,E1 9107.302,E2 9107.302} C_VEL
LIN {X 0,Y 570.485,Z 948.94,A -85,B 0,C 180,E1 9107.938,E2 9107.938} C_VEL
LIN {X 0,Y 570.043,Z 948.94,A -85,B 0,C 180,E1 9117.719,E2 9117.719} C_VEL
LIN {X 0,Y 569.901,Z 948.94,A -85,B 0,C 180,E1 9126.753,E2 9126.753} C_VEL
LIN {X 0,Y 570.001,Z 948.94,A -85,B 0,C 180,E1 9135.097,E2 9135.097} C_VEL
LIN {X 0,Y 569.987,Z 948.94,A -85,B 0,C 180,E1 9144.216,E2 9144.216} C_VEL
LIN {X 0,Y 570.122,Z 948.94,A -85,B 0,C 180,E1 9152.984,E2 9152.984} C_VEL
LIN {X 0,Y 570.36,Z 948.94,A -85,B 0,C 180,E1 9162.164,E2 9162.164} C_VEL
LIN {X 0,Y 570.964,Z 948.94,A -85,B 0,C 180,E1 9170.035,E2 9170.035} C_VEL
LIN {X 0,Y 570.652,Z 948.94,A -85,B 0,C 180,E1 9179.223,E2 9179.223} C_VEL
LIN {X 0,Y 570.592,Z 948.94,A -85,B 0,C 180,E1 9186.86,E2 9186.86} C_VEL
LIN {X 0,Y 570.396,Z 948.94,A -85,B 0,C 180,E1 9194.627,E2 9194.627} C_VEL
LIN {X 0,Y 569.984,Z 948.94,A -85,B 0,C 180,E1 9203.406,E2 9203.406} C_VEL
LIN {X 0,Y 570.341,Z 948.94,A -85,B 0,C 180,E1 9211.244,E2 9211.244} C_VEL
LIN {X 0,Y 570.172,Z 948.94,A -85,B 0,C 180,E1 9220.734,E2 9220.734} C_VEL
LIN {X 0,Y 570.118,Z 948.94,A -85,B 0,C 180,E1 9229.355,E2 9229.355} C_VEL
LIN {X 0,Y 570.534,Z 950.362,A -85,B 0,C 180,E1 9233.19,E2 9233.19} C_VEL
LIN {X 0,Y 595.738,Z 1017.132,A -85,B 0,C 180,E1 9236.4,E2 9236.4} C_VEL
LIN {X 0,Y 592.566,Z 1056.156,A -85,B 0,C 180,E1 9237.446,E2 9237.446} C_VEL
LIN {X 0,Y 582.664,Z 1088.92,A -85,B 0,C 180,E1 9238.367,E2 9238.367} C_VEL
LIN {X 0,Y 575.56,Z 1155.395,A -85,B 0,C 180,E1 9242.249,E2 9242.249} C_VEL
LIN {X 0,Y 569.56,Z 1211.064,A -85,B 0,C 180,E1 9247.318,E2 9247.318} C_VEL
LIN {X 0,Y 565.615,Z 1253.987,A -85,B 0,C 180,E1 9253.279,E2 9253.279} C_VEL
LIN {X 0,Y 563.881,Z 1282.173,A -85,B 0,C 180,E1 9259.593,E2 9259.593} C_VEL
LIN {X 0,Y 563.553,Z 1296.753,A -85,B 0,C 180,E1 9266.179,E2 9266.179} C_VEL
LIN {X 0,Y 563.355,Z 1297.959,A -85,B 0,C 180,E1 9272.353,E2 9272.353} C_VEL
LIN {X 0,Y 563.397,Z 1287.138,A -85,B 0,C 180,E1 9278.556,E2 9278.556} C_VEL
LIN {X 0,Y 564.519,Z 1263.947,A -85,B 0,C 180,E1 9284.42,E2 9284.42} C_VEL
LIN {X 0,Y 567.1,Z 1227.42,A -85,B 0,C 180,E1 9289.893,E2 9289.893} C_VEL
LIN {X 0,Y 570.916,Z 1176.269,A -85,B 0,C 180,E1 9294.783,E2 9294.783} C_VEL
LIN {X 0,Y 575.284,Z 1108.858,A -85,B 0,C 180,E1 9298.922,E2 9298.922} C_VEL
LIN {X 0,Y 579.735,Z 1030.039,A -85,B 0,C 180,E1 9301.884,E2 9301.884} C_VEL
LIN {X 0,Y 578.581,Z 1004.159,A -85,B 0,C 180,E1 9302.635,E2 9302.635} C_VEL
LIN {X 0,Y 562.01,Z 948.94,A -85,B 0,C 180,E1 9304.772,E2 9304.772} C_VEL
LIN {X 0,Y 561.895,Z 948.94,A -85,B 0,C 180,E1 9314.311,E2 9314.311} C_VEL
LIN {X 0,Y 562.172,Z 950.169,A -85,B 0,C 180,E1 9323.059,E2 9323.059} C_VEL
LIN {X 0,Y 581.677,Z 1013.239,A -85,B 0,C 180,E1 9325.392,E2 9325.392} C_VEL
LIN {X 0,Y 577.842,Z 1074.636,A -85,B 0,C 180,E1 9328.14,E2 9328.14} C_VEL
LIN {X 0,Y 572.645,Z 1128.946,A -85,B 0,C 180,E1 9332.274,E2 9332.274} C_VEL
LIN {X 0,Y 567.897,Z 1173.63,A -85,B 0,C 180,E1 9337.629,E2 9337.629} C_VEL
LIN {X 0,Y 564.634,Z 1206.862,A -85,B 0,C 180,E1 9344.022,E2 9344.022} C_VEL
LIN {X 0,Y 563.229,Z 1225.664,A -85,B 0,C 180,E1 9350.71,E2 9350.71} C_VEL
LIN {X 0,Y 562.98,Z 1231.033,A -85,B 0,C 180,E1 9356.15,E2 9356.15} C_VEL
LIN {X 0,Y 563.027,Z 1227.007,A -85,B 0,C 180,E1 9362.333,E2 9362.333} C_VEL
LIN {X 0,Y 564.235,Z 1210.373,A -85,B 0,C 180,E1 9368.913,E2 9368.913} C_VEL
LIN {X 0,Y 567.261,Z 1178.496,A -85,B 0,C 180,E1 9375.539,E2 9375.539} C_VEL
LIN {X 0,Y 572.436,Z 1134.079,A -85,B 0,C 180,E1 9381.258,E2 9381.258} C_VEL
LIN {X 0,Y 578.578,Z 1079.801,A -85,B 0,C 180,E1 9385.769,E2 9385.769} C_VEL
LIN {X 0,Y 584.312,Z 1016.677,A -85,B 0,C 180,E1 9388.987,E2 9388.987} C_VEL
LIN {X 0,Y 581.029,Z 996.197,A -85,B 0,C 180,E1 9389.942,E2 9389.942} C_VEL
LIN {X 0,Y 561.894,Z 948.94,A -85,B 0,C 180,E1 9392.371,E2 9392.371} C_VEL
LIN {X 0,Y 561.688,Z 948.94,A -85,B 0,C 180,E1 9401.476,E2 9401.476} C_VEL
LIN {X 0,Y 561.952,Z 948.94,A -85,B 0,C 180,E1 9410.568,E2 9410.568} C_VEL
LIN {X 0,Y 562.093,Z 948.94,A -85,B 0,C 180,E1 9419.997,E2 9419.997} C_VEL
LIN {X 0,Y 562.503,Z 949.18,A -85,B 0,C 180,E1 9429.715,E2 9429.715} C_VEL
LIN {X 0,Y 571.751,Z 989.555,A -85,B 0,C 180,E1 9430.587,E2 9430.587} C_VEL
LIN {X 0,Y 571.219,Z 1044.4,A -85,B 0,C 180,E1 9431.764,E2 9431.764} C_VEL
LIN {X 0,Y 569.025,Z 1090.105,A -85,B 0,C 180,E1 9434.298,E2 9434.298} C_VEL
LIN {X 0,Y 566.573,Z 1126.416,A -85,B 0,C 180,E1 9438.082,E2 9438.082} C_VEL
LIN {X 0,Y 564.883,Z 1149.973,A -85,B 0,C 180,E1 9442.632,E2 9442.632} C_VEL
LIN {X 0,Y 564.065,Z 1160.279,A -85,B 0,C 180,E1 9447.65,E2 9447.65} C_VEL
LIN {X 0,Y 564.175,Z 1157.78,A -85,B 0,C 180,E1 9452.274,E2 9452.274} C_VEL
LIN {X 0,Y 565.174,Z 1141.323,A -85,B 0,C 180,E1 9457.288,E2 9457.288} C_VEL
LIN {X 0,Y 567.233,Z 1111.252,A -85,B 0,C 180,E1 9461.647,E2 9461.647} C_VEL
LIN {X 0,Y 569.897,Z 1069.902,A -85,B 0,C 180,E1 9464.907,E2 9464.907} C_VEL
LIN {X 0,Y 571.64,Z 1021.804,A -85,B 0,C 180,E1 9466.762,E2 9466.762} C_VEL
LIN {X 0,Y 569.443,Z 974.267,A -85,B 0,C 180,E1 9467.541,E2 9467.541} C_VEL
LIN {X 0,Y 562.474,Z 948.94,A -85,B 0,C 180,E1 9468.192,E2 9468.192} C_VEL
LIN {X 0,Y 561.987,Z 948.94,A -85,B 0,C 180,E1 9478.151,E2 9478.151} C_VEL
LIN {X 0,Y 561.844,Z 948.94,A -85,B 0,C 180,E1 9487.369,E2 9487.369} C_VEL
LIN {X 0,Y 561.948,Z 948.94,A -85,B 0,C 180,E1 9496.448,E2 9496.448} C_VEL
LIN {X 0,Y 561.963,Z 948.94,A -85,B 0,C 180,E1 9505.368,E2 9505.368} C_VEL
LIN {X 0,Y 562.132,Z 948.94,A -85,B 0,C 180,E1 9514.628,E2 9514.628} C_VEL
LIN {X 0,Y 562.544,Z 948.94,A -85,B 0,C 180,E1 9523.527,E2 9523.527} C_VEL
LIN {X 0,Y 562.608,Z 948.94,A -85,B 0,C 180,E1 9531.452,E2 9531.452} C_VEL
LIN {X 0,Y 562.653,Z 948.94,A -85,B 0,C 180,E1 9539.212,E2 9539.212} C_VEL
LIN {X 0,Y 562.563,Z 948.94,A -85,B 0,C 180,E1 9546.958,E2 9546.958} C_VEL
LIN {X 0,Y 562.334,Z 948.94,A -85,B 0,C 180,E1 9554.842,E2 9554.842} C_VEL
LIN {X 0,Y 562.046,Z 948.94,A -85,B 0,C 180,E1 9563.036,E2 9563.036} C_VEL
LIN {X 0,Y 562.285,Z 948.94,A -85,B 0,C 180,E1 9571.861,E2 9571.861} C_VEL
LIN {X 0,Y 562.08,Z 948.94,A -85,B 0,C 180,E1 9581.4,E2 9581.4} C_VEL
LIN {X 0,Y 562.129,Z 948.94,A -85,B 0,C 180,E1 9590.681,E2 9590.681} C_VEL
LIN {X 0,Y 562.654,Z 951.17,A -85,B 0,C 180,E1 9592.813,E2 9592.813} C_VEL
LIN {X 0,Y 588.803,Z 1020.612,A -85,B 0,C 180,E1 9596.06,E2 9596.06} C_VEL
LIN {X 0,Y 582.664,Z 1088.92,A -85,B 0,C 180,E1 9598.367,E2 9598.367} C_VEL
LIN {X 0,Y 571.907,Z 1120.278,A -85,B 0,C 180,E1 9599.625,E2 9599.625} C_VEL
LIN {X 0,Y 565.079,Z 1182.368,A -85,B 0,C 180,E1 9604.186,E2 9604.186} C_VEL
LIN {X 0,Y 559.751,Z 1233.465,A -85,B 0,C 180,E1 9609.948,E2 9609.948} C_VEL
LIN {X 0,Y 556.517,Z 1269.458,A -85,B 0,C 180,E1 9616.275,E2 9616.275} C_VEL
LIN {X 0,Y 555.38,Z 1289.311,A -85,B 0,C 180,E1 9622.188,E2 9622.188} C_VEL
LIN {X 0,Y 555.164,Z 1297.665,A -85,B 0,C 180,E1 9627.689,E2 9627.689} C_VEL
LIN {X 0,Y 555.074,Z 1295.87,A -85,B 0,C 180,E1 9633.957,E2 9633.957} C_VEL
LIN {X 0,Y 555.475,Z 1282.653,A -85,B 0,C 180,E1 9639.869,E2 9639.869} C_VEL
LIN {X 0,Y 556.943,Z 1257.057,A -85,B 0,C 180,E1 9645.646,E2 9645.646} C_VEL
LIN {X 0,Y 559.779,Z 1218.216,A -85,B 0,C 180,E1 9650.994,E2 9650.994} C_VEL
LIN {X 0,Y 563.747,Z 1164.232,A -85,B 0,C 180,E1 9655.79,E2 9655.79} C_VEL
LIN {X 0,Y 568.333,Z 1093.986,A -85,B 0,C 180,E1 9659.809,E2 9659.809} C_VEL
LIN {X 0,Y 571.923,Z 1008.323,A -85,B 0,C 180,E1 9662.788,E2 9662.788} C_VEL
LIN {X 0,Y 553.994,Z 948.94,A -85,B 0,C 180,E1 9665.239,E2 9665.239} C_VEL
LIN {X 0,Y 553.89,Z 948.94,A -85,B 0,C 180,E1 9674.362,E2 9674.362} C_VEL
LIN {X 0,Y 554.123,Z 950.24,A -85,B 0,C 180,E1 9682.59,E2 9682.59} C_VEL
LIN {X 0,Y 574.491,Z 1014.339,A -85,B 0,C 180,E1 9685.062,E2 9685.062} C_VEL
LIN {X 0,Y 570.653,Z 1074.528,A -85,B 0,C 180,E1 9687.768,E2 9687.768} C_VEL
LIN {X 0,Y 565.427,Z 1127.643,A -85,B 0,C 180,E1 9691.8,E2 9691.8} C_VEL
LIN {X 0,Y 560.405,Z 1172.55,A -85,B 0,C 180,E1 9697.145,E2 9697.145} C_VEL
LIN {X 0,Y 557.049,Z 1205.484,A -85,B 0,C 180,E1 9703.392,E2 9703.392} C_VEL
LIN {X 0,Y 555.56,Z 1224.564,A -85,B 0,C 180,E1 9709.787,E2 9709.787} C_VEL
LIN {X 0,Y 555.002,Z 1231.664,A -85,B 0,C 180,E1 9716.874,E2 9716.874} C_VEL
LIN {X 0,Y 555.557,Z 1224.757,A -85,B 0,C 180,E1 9723.932,E2 9723.932} C_VEL
LIN {X 0,Y 557.185,Z 1204.327,A -85,B 0,C 180,E1 9730.749,E2 9730.749} C_VEL
LIN {X 0,Y 560.766,Z 1168.883,A -85,B 0,C 180,E1 9737.337,E2 9737.337} C_VEL
LIN {X 0,Y 566.666,Z 1121.293,A -85,B 0,C 180,E1 9742.87,E2 9742.87} C_VEL
LIN {X 0,Y 573.026,Z 1064.789,A -85,B 0,C 180,E1 9747.082,E2 9747.082} C_VEL
LIN {X 0,Y 576.272,Z 1005.486,A -85,B 0,C 180,E1 9749.892,E2 9749.892} C_VEL
LIN {X 0,Y 553.852,Z 948.94,A -85,B 0,C 180,E1 9752.817,E2 9752.817} C_VEL
LIN {X 0,Y 553.709,Z 948.94,A -85,B 0,C 180,E1 9762.21,E2 9762.21} C_VEL
LIN {X 0,Y 553.957,Z 948.94,A -85,B 0,C 180,E1 9771.907,E2 9771.907} C_VEL
LIN {X 0,Y 554.063,Z 948.94,A -85,B 0,C 180,E1 9781.321,E2 9781.321} C_VEL
LIN {X 0,Y 554.556,Z 949.994,A -85,B 0,C 180,E1 9789.422,E2 9789.422} C_VEL
LIN {X 0,Y 564.232,Z 989.617,A -85,B 0,C 180,E1 9790.318,E2 9790.318} C_VEL
LIN {X 0,Y 563.663,Z 1045.053,A -85,B 0,C 180,E1 9791.511,E2 9791.511} C_VEL
LIN {X 0,Y 561.365,Z 1090.914,A -85,B 0,C 180,E1 9794.077,E2 9794.077} C_VEL
LIN {X 0,Y 558.908,Z 1126.228,A -85,B 0,C 180,E1 9797.766,E2 9797.766} C_VEL
LIN {X 0,Y 557.004,Z 1150.892,A -85,B 0,C 180,E1 9802.527,E2 9802.527} C_VEL
LIN {X 0,Y 556.149,Z 1161.223,A -85,B 0,C 180,E1 9807.616,E2 9807.616} C_VEL
LIN {X 0,Y 556.253,Z 1158.75,A -85,B 0,C 180,E1 9812.306,E2 9812.306} C_VEL
LIN {X 0,Y 557.321,Z 1142.318,A -85,B 0,C 180,E1 9817.391,E2 9817.391} C_VEL
LIN {X 0,Y 559.493,Z 1112.287,A -85,B 0,C 180,E1 9821.81,E2 9821.81} C_VEL
LIN {X 0,Y 562.267,Z 1070.996,A -85,B 0,C 180,E1 9825.115,E2 9825.115} C_VEL
LIN {X 0,Y 564.075,Z 1022.35,A -85,B 0,C 180,E1 9827.011,E2 9827.011} C_VEL
LIN {X 0,Y 561.918,Z 976.022,A -85,B 0,C 180,E1 9827.781,E2 9827.781} C_VEL
LIN {X 0,Y 554.469,Z 948.94,A -85,B 0,C 180,E1 9828.507,E2 9828.507} C_VEL
LIN {X 0,Y 553.999,Z 948.94,A -85,B 0,C 180,E1 9838.594,E2 9838.594} C_VEL
LIN {X 0,Y 553.737,Z 948.94,A -85,B 0,C 180,E1 9848.013,E2 9848.013} C_VEL
LIN {X 0,Y 553.942,Z 948.94,A -85,B 0,C 180,E1 9857.812,E2 9857.812} C_VEL
LIN {X 0,Y 554.034,Z 948.94,A -85,B 0,C 180,E1 9867.691,E2 9867.691} C_VEL
LIN {X 0,Y 554.259,Z 948.94,A -85,B 0,C 180,E1 9876.588,E2 9876.588} C_VEL
LIN {X 0,Y 555.037,Z 948.94,A -85,B 0,C 180,E1 9886.543,E2 9886.543} C_VEL
LIN {X 0,Y 555.053,Z 948.94,A -85,B 0,C 180,E1 9896.763,E2 9896.763} C_VEL
LIN {X 0,Y 554.976,Z 948.94,A -85,B 0,C 180,E1 9905.477,E2 9905.477} C_VEL
LIN {X 0,Y 554.278,Z 948.94,A -85,B 0,C 180,E1 9915.063,E2 9915.063} C_VEL
LIN {X 0,Y 553.96,Z 948.94,A -85,B 0,C 180,E1 9923.527,E2 9923.527} C_VEL
LIN {X 0,Y 554.255,Z 948.94,A -85,B 0,C 180,E1 9932.258,E2 9932.258} C_VEL
LIN {X 0,Y 554.055,Z 948.94,A -85,B 0,C 180,E1 9942.136,E2 9942.136} C_VEL
LIN {X 0,Y 554.43,Z 950.271,A -85,B 0,C 180,E1 9952.18,E2 9952.18} C_VEL
LIN {X 0,Y 581.806,Z 1022.623,A -85,B 0,C 180,E1 9955.695,E2 9955.695} C_VEL
LIN {X 0,Y 575.052,Z 1093.124,A -85,B 0,C 180,E1 9958.194,E2 9958.194} C_VEL
LIN {X 0,Y 571.907,Z 1120.278,A -85,B 0,C 180,E1 9959.625,E2 9959.625} C_VEL
LIN {X 0,Y 561.223,Z 1150.04,A -85,B 0,C 180,E1 9961.26,E2 9961.26} C_VEL
LIN {X 0,Y 554.427,Z 1207.297,A -85,B 0,C 180,E1 9966.467,E2 9966.467} C_VEL
LIN {X 0,Y 549.983,Z 1250.097,A -85,B 0,C 180,E1 9972.376,E2 9972.376} C_VEL
LIN {X 0,Y 547.823,Z 1279.529,A -85,B 0,C 180,E1 9978.843,E2 9978.843} C_VEL
LIN {X 0,Y 547.414,Z 1295.222,A -85,B 0,C 180,E1 9985.619,E2 9985.619} C_VEL
LIN {X 0,Y 547.379,Z 1296.946,A -85,B 0,C 180,E1 9992.422,E2 9992.422} C_VEL
LIN {X 0,Y 547.417,Z 1285.556,A -85,B 0,C 180,E1 9998.808,E2 9998.808} C_VEL
LIN {X 0,Y 548.546,Z 1262.367,A -85,B 0,C 180,E1 10004.656,E2 10004.656} C_VEL
LIN {X 0,Y 551.261,Z 1225.788,A -85,B 0,C 180,E1 10010.165,E2 10010.165} C_VEL
LIN {X 0,Y 555.138,Z 1174.859,A -85,B 0,C 180,E1 10015.107,E2 10015.107} C_VEL
LIN {X 0,Y 559.86,Z 1106.597,A -85,B 0,C 180,E1 10019.408,E2 10019.408} C_VEL
LIN {X 0,Y 564.976,Z 1025.765,A -85,B 0,C 180,E1 10022.557,E2 10022.557} C_VEL
LIN {X 0,Y 563.216,Z 1007.008,A -85,B 0,C 180,E1 10023.194,E2 10023.194} C_VEL
LIN {X 0,Y 547.319,Z 953.36,A -85,B 0,C 180,E1 10025.438,E2 10025.438} C_VEL
LIN {X 0,Y 545.97,Z 948.94,A -85,B 0,C 180,E1 10025.907,E2 10025.907} C_VEL
LIN {X 0,Y 545.87,Z 948.94,A -85,B 0,C 180,E1 10035.192,E2 10035.192} C_VEL
LIN {X 0,Y 545.911,Z 949.418,A -85,B 0,C 180,E1 10042.059,E2 10042.059} C_VEL
LIN {X 0,Y 567.423,Z 1013.762,A -85,B 0,C 180,E1 10044.667,E2 10044.667} C_VEL
LIN {X 0,Y 563.556,Z 1073.341,A -85,B 0,C 180,E1 10047.311,E2 10047.311} C_VEL
LIN {X 0,Y 558.097,Z 1127.485,A -85,B 0,C 180,E1 10051.417,E2 10051.417} C_VEL
LIN {X 0,Y 552.752,Z 1172.784,A -85,B 0,C 180,E1 10056.844,E2 10056.844} C_VEL
LIN {X 0,Y 548.996,Z 1207.363,A -85,B 0,C 180,E1 10063.554,E2 10063.554} C_VEL
LIN {X 0,Y 547.328,Z 1226.655,A -85,B 0,C 180,E1 10070.55,E2 10070.55} C_VEL
LIN {X 0,Y 547.089,Z 1232.007,A -85,B 0,C 180,E1 10077.631,E2 10077.631} C_VEL
LIN {X 0,Y 547.921,Z 1223.711,A -85,B 0,C 180,E1 10084.783,E2 10084.783} C_VEL
LIN {X 0,Y 549.399,Z 1200.398,A -85,B 0,C 180,E1 10091.974,E2 10091.974} C_VEL
LIN {X 0,Y 553.61,Z 1163.729,A -85,B 0,C 180,E1 10098.395,E2 10098.395} C_VEL
LIN {X 0,Y 560.065,Z 1115.164,A -85,B 0,C 180,E1 10103.79,E2 10103.79} C_VEL
LIN {X 0,Y 566.667,Z 1057.218,A -85,B 0,C 180,E1 10107.908,E2 10107.908} C_VEL
LIN {X 0,Y 569.55,Z 1009.062,A -85,B 0,C 180,E1 10110.142,E2 10110.142} C_VEL
LIN {X 0,Y 545.799,Z 948.94,A -85,B 0,C 180,E1 10113.363,E2 10113.363} C_VEL
LIN {X 0,Y 545.75,Z 948.94,A -85,B 0,C 180,E1 10122.973,E2 10122.973} C_VEL
LIN {X 0,Y 545.931,Z 948.94,A -85,B 0,C 180,E1 10132.432,E2 10132.432} C_VEL
LIN {X 0,Y 546.053,Z 948.94,A -85,B 0,C 180,E1 10141.145,E2 10141.145} C_VEL
LIN {X 0,Y 546.589,Z 950.131,A -85,B 0,C 180,E1 10149.108,E2 10149.108} C_VEL
LIN {X 0,Y 556.726,Z 992.086,A -85,B 0,C 180,E1 10150.074,E2 10150.074} C_VEL
LIN {X 0,Y 556.036,Z 1048.057,A -85,B 0,C 180,E1 10151.339,E2 10151.339} C_VEL
LIN {X 0,Y 553.659,Z 1092.511,A -85,B 0,C 180,E1 10153.915,E2 10153.915} C_VEL
LIN {X 0,Y 550.953,Z 1128.872,A -85,B 0,C 180,E1 10157.839,E2 10157.839} C_VEL
LIN {X 0,Y 549.121,Z 1151.811,A -85,B 0,C 180,E1 10162.419,E2 10162.419} C_VEL
LIN {X 0,Y 548.233,Z 1162.167,A -85,B 0,C 180,E1 10167.582,E2 10167.582} C_VEL
LIN {X 0,Y 548.326,Z 1159.72,A -85,B 0,C 180,E1 10172.34,E2 10172.34} C_VEL
LIN {X 0,Y 549.466,Z 1143.313,A -85,B 0,C 180,E1 10177.497,E2 10177.497} C_VEL
LIN {X 0,Y 551.678,Z 1114.376,A -85,B 0,C 180,E1 10181.864,E2 10181.864} C_VEL
LIN {X 0,Y 554.527,Z 1073.727,A -85,B 0,C 180,E1 10185.229,E2 10185.229} C_VEL
LIN {X 0,Y 556.438,Z 1025.152,A -85,B 0,C 180,E1 10187.219,E2 10187.219} C_VEL
LIN {X 0,Y 554.331,Z 977.353,A -85,B 0,C 180,E1 10188.037,E2 10188.037} C_VEL
LIN {X 0,Y 546.475,Z 948.94,A -85,B 0,C 180,E1 10188.765,E2 10188.765} C_VEL
LIN {X 0,Y 545.932,Z 948.94,A -85,B 0,C 180,E1 10199.057,E2 10199.057} C_VEL
LIN {X 0,Y 545.737,Z 948.94,A -85,B 0,C 180,E1 10208.672,E2 10208.672} C_VEL
LIN {X 0,Y 545.939,Z 948.94,A -85,B 0,C 180,E1 10217.375,E2 10217.375} C_VEL
LIN {X 0,Y 546.003,Z 948.94,A -85,B 0,C 180,E1 10227.157,E2 10227.157} C_VEL
LIN {X 0,Y 546.209,Z 948.94,A -85,B 0,C 180,E1 10236.222,E2 10236.222} C_VEL
LIN {X 0,Y 547.014,Z 948.94,A -85,B 0,C 180,E1 10246.342,E2 10246.342} C_VEL
LIN {X 0,Y 547.055,Z 948.94,A -85,B 0,C 180,E1 10256.775,E2 10256.775} C_VEL
LIN {X 0,Y 546.939,Z 948.94,A -85,B 0,C 180,E1 10265.558,E2 10265.558} C_VEL
LIN {X 0,Y 546.225,Z 948.94,A -85,B 0,C 180,E1 10275.29,E2 10275.29} C_VEL
LIN {X 0,Y 545.94,Z 948.94,A -85,B 0,C 180,E1 10283.757,E2 10283.757} C_VEL
LIN {X 0,Y 546.268,Z 948.94,A -85,B 0,C 180,E1 10292.788,E2 10292.788} C_VEL
LIN {X 0,Y 546.023,Z 948.94,A -85,B 0,C 180,E1 10302.635,E2 10302.635} C_VEL
LIN {X 0,Y 546.48,Z 950.944,A -85,B 0,C 180,E1 10311.592,E2 10311.592} C_VEL
LIN {X 0,Y 574.978,Z 1022.994,A -85,B 0,C 180,E1 10315.285,E2 10315.285} C_VEL
LIN {X 0,Y 567.802,Z 1093.905,A -85,B 0,C 180,E1 10317.864,E2 10317.864} C_VEL
LIN {X 0,Y 561.223,Z 1150.04,A -85,B 0,C 180,E1 10321.26,E2 10321.26} C_VEL
LIN {X 0,Y 550.369,Z 1177.859,A -85,B 0,C 180,E1 10323.243,E2 10323.243} C_VEL
LIN {X 0,Y 544.35,Z 1230.029,A -85,B 0,C 180,E1 10329.127,E2 10329.127} C_VEL
LIN {X 0,Y 540.831,Z 1267.801,A -85,B 0,C 180,E1 10335.794,E2 10335.794} C_VEL
LIN {X 0,Y 539.474,Z 1288.256,A -85,B 0,C 180,E1 10341.956,E2 10341.956} C_VEL
LIN {X 0,Y 539.21,Z 1296.723,A -85,B 0,C 180,E1 10347.621,E2 10347.621} C_VEL
LIN {X 0,Y 539.305,Z 1296.186,A -85,B 0,C 180,E1 10352.776,E2 10352.776} C_VEL
LIN {X 0,Y 539.439,Z 1283.753,A -85,B 0,C 180,E1 10359.288,E2 10359.288} C_VEL
LIN {X 0,Y 540.703,Z 1259.336,A -85,B 0,C 180,E1 10365.204,E2 10365.204} C_VEL
LIN {X 0,Y 543.582,Z 1221.396,A -85,B 0,C 180,E1 10370.752,E2 10370.752} C_VEL
LIN {X 0,Y 547.784,Z 1167.522,A -85,B 0,C 180,E1 10375.81,E2 10375.81} C_VEL
LIN {X 0,Y 552.664,Z 1097.71,A -85,B 0,C 180,E1 10380.059,E2 10380.059} C_VEL
LIN {X 0,Y 556.764,Z 1011.759,A -85,B 0,C 180,E1 10383.336,E2 10383.336} C_VEL
LIN {X 0,Y 540.917,Z 957.167,A -85,B 0,C 180,E1 10385.773,E2 10385.773} C_VEL
LIN {X 0,Y 537.926,Z 948.94,A -85,B 0,C 180,E1 10386.209,E2 10386.209} C_VEL
LIN {X 0,Y 537.756,Z 948.94,A -85,B 0,C 180,E1 10396.069,E2 10396.069} C_VEL
LIN {X 0,Y 538.087,Z 950.859,A -85,B 0,C 180,E1 10401.542,E2 10401.542} C_VEL
LIN {X 0,Y 559.267,Z 1012.11,A -85,B 0,C 180,E1 10404.151,E2 10404.151} C_VEL
LIN {X 0,Y 556.516,Z 1072.876,A -85,B 0,C 180,E1 10406.882,E2 10406.882} C_VEL
LIN {X 0,Y 550.791,Z 1127.531,A -85,B 0,C 180,E1 10411.035,E2 10411.035} C_VEL
LIN {X 0,Y 545.146,Z 1172.797,A -85,B 0,C 180,E1 10416.502,E2 10416.502} C_VEL
LIN {X 0,Y 541.44,Z 1205.919,A -85,B 0,C 180,E1 10422.898,E2 10422.898} C_VEL
LIN {X 0,Y 539.701,Z 1225.349,A -85,B 0,C 180,E1 10429.483,E2 10429.483} C_VEL
LIN {X 0,Y 539.051,Z 1232.462,A -85,B 0,C 180,E1 10435.979,E2 10435.979} C_VEL
LIN {X 0,Y 539.125,Z 1228.533,A -85,B 0,C 180,E1 10442.436,E2 10442.436} C_VEL
LIN {X 0,Y 540.577,Z 1211.969,A -85,B 0,C 180,E1 10449.307,E2 10449.307} C_VEL
LIN {X 0,Y 544.124,Z 1180.106,A -85,B 0,C 180,E1 10456.214,E2 10456.214} C_VEL
LIN {X 0,Y 549.831,Z 1136.487,A -85,B 0,C 180,E1 10462.067,E2 10462.067} C_VEL
LIN {X 0,Y 556.804,Z 1082.361,A -85,B 0,C 180,E1 10466.747,E2 10466.747} C_VEL
LIN {X 0,Y 563.123,Z 1020.561,A -85,B 0,C 180,E1 10470.039,E2 10470.039} C_VEL
LIN {X 0,Y 555.143,Z 990.598,A -85,B 0,C 180,E1 10471.661,E2 10471.661} C_VEL
LIN {X 0,Y 537.795,Z 948.94,A -85,B 0,C 180,E1 10473.99,E2 10473.99} C_VEL
LIN {X 0,Y 537.705,Z 948.94,A -85,B 0,C 180,E1 10483.926,E2 10483.926} C_VEL
LIN {X 0,Y 537.87,Z 948.94,A -85,B 0,C 180,E1 10493.563,E2 10493.563} C_VEL
LIN {X 0,Y 538.051,Z 948.94,A -85,B 0,C 180,E1 10502.731,E2 10502.731} C_VEL
LIN {X 0,Y 538.494,Z 949.767,A -85,B 0,C 180,E1 10508.773,E2 10508.773} C_VEL
LIN {X 0,Y 549.212,Z 992.995,A -85,B 0,C 180,E1 10509.801,E2 10509.801} C_VEL
LIN {X 0,Y 548.489,Z 1048.719,A -85,B 0,C 180,E1 10511.072,E2 10511.072} C_VEL
LIN {X 0,Y 546.033,Z 1093.168,A -85,B 0,C 180,E1 10513.67,E2 10513.67} C_VEL
LIN {X 0,Y 543.194,Z 1129.75,A -85,B 0,C 180,E1 10517.662,E2 10517.662} C_VEL
LIN {X 0,Y 541.251,Z 1152.729,A -85,B 0,C 180,E1 10522.308,E2 10522.308} C_VEL
LIN {X 0,Y 540.317,Z 1163.111,A -85,B 0,C 180,E1 10527.546,E2 10527.546} C_VEL
LIN {X 0,Y 540.405,Z 1160.69,A -85,B 0,C 180,E1 10532.374,E2 10532.374} C_VEL
LIN {X 0,Y 541.61,Z 1144.309,A -85,B 0,C 180,E1 10537.607,E2 10537.607} C_VEL
LIN {X 0,Y 543.917,Z 1115.409,A -85,B 0,C 180,E1 10542.036,E2 10542.036} C_VEL
LIN {X 0,Y 546.899,Z 1074.819,A -85,B 0,C 180,E1 10545.447,E2 10545.447} C_VEL
LIN {X 0,Y 548.859,Z 1026.398,A -85,B 0,C 180,E1 10547.466,E2 10547.466} C_VEL
LIN {X 0,Y 546.828,Z 978.937,A -85,B 0,C 180,E1 10548.293,E2 10548.293} C_VEL
LIN {X 0,Y 538.405,Z 948.94,A -85,B 0,C 180,E1 10549.15,E2 10549.15} C_VEL
LIN {X 0,Y 537.848,Z 948.94,A -85,B 0,C 180,E1 10559.536,E2 10559.536} C_VEL
LIN {X 0,Y 537.691,Z 948.94,A -85,B 0,C 180,E1 10569.362,E2 10569.362} C_VEL
LIN {X 0,Y 537.839,Z 948.94,A -85,B 0,C 180,E1 10578.436,E2 10578.436} C_VEL
LIN {X 0,Y 537.905,Z 948.94,A -85,B 0,C 180,E1 10586.598,E2 10586.598} C_VEL
LIN {X 0,Y 538.203,Z 948.94,A -85,B 0,C 180,E1 10596.28,E2 10596.28} C_VEL
LIN {X 0,Y 538.971,Z 948.94,A -85,B 0,C 180,E1 10606.134,E2 10606.134} C_VEL
LIN {X 0,Y 539.086,Z 948.94,A -85,B 0,C 180,E1 10616.818,E2 10616.818} C_VEL
LIN {X 0,Y 538.921,Z 948.94,A -85,B 0,C 180,E1 10625.641,E2 10625.641} C_VEL
LIN {X 0,Y 538.19,Z 948.94,A -85,B 0,C 180,E1 10635.524,E2 10635.524} C_VEL
LIN {X 0,Y 537.905,Z 948.94,A -85,B 0,C 180,E1 10644.134,E2 10644.134} C_VEL
LIN {X 0,Y 538.173,Z 948.94,A -85,B 0,C 180,E1 10653.799,E2 10653.799} C_VEL
LIN {X 0,Y 537.971,Z 948.94,A -85,B 0,C 180,E1 10661.695,E2 10661.695} C_VEL
LIN {X 0,Y 538.368,Z 950.897,A -85,B 0,C 180,E1 10670.956,E2 10670.956} C_VEL
LIN {X 0,Y 568.016,Z 1023.982,A -85,B 0,C 180,E1 10674.878,E2 10674.878} C_VEL
LIN {X 0,Y 560.691,Z 1093.753,A -85,B 0,C 180,E1 10677.484,E2 10677.484} C_VEL
LIN {X 0,Y 552.573,Z 1159.244,A -85,B 0,C 180,E1 10681.661,E2 10681.661} C_VEL
LIN {X 0,Y 550.369,Z 1177.859,A -85,B 0,C 180,E1 10683.243,E2 10683.243} C_VEL
LIN {X 0,Y 539.337,Z 1203.376,A -85,B 0,C 180,E1 10685.568,E2 10685.568} C_VEL
LIN {X 0,Y 534.368,Z 1247.104,A -85,B 0,C 180,E1 10691.616,E2 10691.616} C_VEL
LIN {X 0,Y 531.916,Z 1276.938,A -85,B 0,C 180,E1 10698.106,E2 10698.106} C_VEL
LIN {X 0,Y 531.223,Z 1292.576,A -85,B 0,C 180,E1 10704.303,E2 10704.303} C_VEL
LIN {X 0,Y 531.594,Z 1296.857,A -85,B 0,C 180,E1 10710.858,E2 10710.858} C_VEL
LIN {X 0,Y 531.56,Z 1287.333,A -85,B 0,C 180,E1 10717.833,E2 10717.833} C_VEL
LIN {X 0,Y 532.564,Z 1265.086,A -85,B 0,C 180,E1 10724.056,E2 10724.056} C_VEL
LIN {X 0,Y 535.117,Z 1228.568,A -85,B 0,C 180,E1 10729.935,E2 10729.935} C_VEL
LIN {X 0,Y 539.221,Z 1177.917,A -85,B 0,C 180,E1 10735.121,E2 10735.121} C_VEL
LIN {X 0,Y 544.191,Z 1109.992,A -85,B 0,C 180,E1 10739.662,E2 10739.662} C_VEL
LIN {X 0,Y 550.05,Z 1027.518,A -85,B 0,C 180,E1 10743.123,E2 10743.123} C_VEL
LIN {X 0,Y 547.501,Z 1008.097,A -85,B 0,C 180,E1 10743.894,E2 10743.894} C_VEL
LIN {X 0,Y 534.934,Z 961.677,A -85,B 0,C 180,E1 10746.063,E2 10746.063} C_VEL
LIN {X 0,Y 529.85,Z 948.94,A -85,B 0,C 180,E1 10746.994,E2 10746.994} C_VEL
LIN {X 0,Y 529.669,Z 948.94,A -85,B 0,C 180,E1 10756.984,E2 10756.984} C_VEL
LIN {X 0,Y 529.983,Z 950.724,A -85,B 0,C 180,E1 10760.925,E2 10760.925} C_VEL
LIN {X 0,Y 547.605,Z 998.687,A -85,B 0,C 180,E1 10763.036,E2 10763.036} C_VEL
LIN {X 0,Y 552.93,Z 1024.696,A -85,B 0,C 180,E1 10764.215,E2 10764.215} C_VEL
LIN {X 0,Y 548.382,Z 1084.078,A -85,B 0,C 180,E1 10767.151,E2 10767.151} C_VEL
LIN {X 0,Y 542.102,Z 1137.709,A -85,B 0,C 180,E1 10771.658,E2 10771.658} C_VEL
LIN {X 0,Y 536.342,Z 1181.628,A -85,B 0,C 180,E1 10777.557,E2 10777.557} C_VEL
LIN {X 0,Y 532.647,Z 1212.371,A -85,B 0,C 180,E1 10784.31,E2 10784.31} C_VEL
LIN {X 0,Y 531.268,Z 1228.631,A -85,B 0,C 180,E1 10790.976,E2 10790.976} C_VEL
LIN {X 0,Y 531.117,Z 1232.984,A -85,B 0,C 180,E1 10797.559,E2 10797.559} C_VEL
LIN {X 0,Y 532.003,Z 1224.759,A -85,B 0,C 180,E1 10804.926,E2 10804.926} C_VEL
LIN {X 0,Y 533.659,Z 1201.448,A -85,B 0,C 180,E1 10812.333,E2 10812.333} C_VEL
LIN {X 0,Y 538.271,Z 1164.682,A -85,B 0,C 180,E1 10818.938,E2 10818.938} C_VEL
LIN {X 0,Y 545.337,Z 1115.884,A -85,B 0,C 180,E1 10824.474,E2 10824.474} C_VEL
LIN {X 0,Y 552.475,Z 1057.919,A -85,B 0,C 180,E1 10828.666,E2 10828.666} C_VEL
LIN {X 0,Y 554.894,Z 1012.247,A -85,B 0,C 180,E1 10830.881,E2 10830.881} C_VEL
LIN {X 0,Y 529.785,Z 948.94,A -85,B 0,C 180,E1 10834.48,E2 10834.48} C_VEL
LIN {X 0,Y 529.645,Z 948.94,A -85,B 0,C 180,E1 10844.618,E2 10844.618} C_VEL
LIN {X 0,Y 529.857,Z 948.94,A -85,B 0,C 180,E1 10854.004,E2 10854.004} C_VEL
LIN {X 0,Y 530.044,Z 948.94,A -85,B 0,C 180,E1 10863.615,E2 10863.615} C_VEL
LIN {X 0,Y 530.538,Z 950.351,A -85,B 0,C 180,E1 10868.445,E2 10868.445} C_VEL
LIN {X 0,Y 541.715,Z 993.086,A -85,B 0,C 180,E1 10869.509,E2 10869.509} C_VEL
LIN {X 0,Y 540.942,Z 1049.657,A -85,B 0,C 180,E1 10870.809,E2 10870.809} C_VEL
LIN {X 0,Y 538.427,Z 1093.989,A -85,B 0,C 180,E1 10873.432,E2 10873.432} C_VEL
LIN {X 0,Y 535.436,Z 1130.629,A -85,B 0,C 180,E1 10877.481,E2 10877.481} C_VEL
LIN {X 0,Y 533.372,Z 1153.649,A -85,B 0,C 180,E1 10882.194,E2 10882.194} C_VEL
LIN {X 0,Y 532.379,Z 1164.058,A -85,B 0,C 180,E1 10887.51,E2 10887.51} C_VEL
LIN {X 0,Y 532.487,Z 1161.658,A -85,B 0,C 180,E1 10892.409,E2 10892.409} C_VEL
LIN {X 0,Y 533.743,Z 1145.305,A -85,B 0,C 180,E1 10897.72,E2 10897.72} C_VEL
LIN {X 0,Y 536.177,Z 1116.439,A -85,B 0,C 180,E1 10902.212,E2 10902.212} C_VEL
LIN {X 0,Y 539.265,Z 1075.911,A -85,B 0,C 180,E1 10905.671,E2 10905.671} C_VEL
LIN {X 0,Y 541.306,Z 1027.634,A -85,B 0,C 180,E1 10907.72,E2 10907.72} C_VEL
LIN {X 0,Y 539.469,Z 980.969,A -85,B 0,C 180,E1 10908.544,E2 10908.544} C_VEL
LIN {X 0,Y 530.33,Z 948.94,A -85,B 0,C 180,E1 10909.453,E2 10909.453} C_VEL
LIN {X 0,Y 529.803,Z 948.94,A -85,B 0,C 180,E1 10920.031,E2 10920.031} C_VEL
LIN {X 0,Y 529.658,Z 948.94,A -85,B 0,C 180,E1 10927.97,E2 10927.97} C_VEL
LIN {X 0,Y 529.778,Z 948.94,A -85,B 0,C 180,E1 10937.658,E2 10937.658} C_VEL
LIN {X 0,Y 529.913,Z 948.94,A -85,B 0,C 180,E1 10947.559,E2 10947.559} C_VEL
LIN {X 0,Y 530.182,Z 948.94,A -85,B 0,C 180,E1 10957.247,E2 10957.247} C_VEL
LIN {X 0,Y 531.058,Z 948.94,A -85,B 0,C 180,E1 10967.606,E2 10967.606} C_VEL
LIN {X 0,Y 531.218,Z 948.94,A -85,B 0,C 180,E1 10977.528,E2 10977.528} C_VEL
LIN {X 0,Y 530.883,Z 948.94,A -85,B 0,C 180,E1 10985.727,E2 10985.727} C_VEL
LIN {X 0,Y 530.144,Z 948.94,A -85,B 0,C 180,E1 10995.766,E2 10995.766} C_VEL
LIN {X 0,Y 529.862,Z 948.94,A -85,B 0,C 180,E1 11004.524,E2 11004.524} C_VEL
LIN {X 0,Y 530.159,Z 948.94,A -85,B 0,C 180,E1 11013.917,E2 11013.917} C_VEL
LIN {X 0,Y 529.858,Z 948.94,A -85,B 0,C 180,E1 11023.156,E2 11023.156} C_VEL
LIN {X 0,Y 530.254,Z 950.809,A -85,B 0,C 180,E1 11030.311,E2 11030.311} C_VEL
LIN {X 0,Y 557.395,Z 1016.463,A -85,B 0,C 180,E1 11033.947,E2 11033.947} C_VEL
LIN {X 0,Y 560.508,Z 1032.434,A -85,B 0,C 180,E1 11034.682,E2 11034.682} C_VEL
LIN {X 0,Y 552.475,Z 1102.571,A -85,B 0,C 180,E1 11037.58,E2 11037.58} C_VEL
LIN {X 0,Y 544.232,Z 1166.01,A -85,B 0,C 180,E1 11041.912,E2 11041.912} C_VEL
LIN {X 0,Y 539.337,Z 1203.376,A -85,B 0,C 180,E1 11045.568,E2 11045.568} C_VEL
LIN {X 0,Y 528.996,Z 1226.369,A -85,B 0,C 180,E1 11048.252,E2 11048.252} C_VEL
LIN {X 0,Y 525.264,Z 1264.417,A -85,B 0,C 180,E1 11054.913,E2 11054.913} C_VEL
LIN {X 0,Y 523.573,Z 1287.189,A -85,B 0,C 180,E1 11061.71,E2 11061.71} C_VEL
LIN {X 0,Y 523.263,Z 1295.776,A -85,B 0,C 180,E1 11067.548,E2 11067.548} C_VEL
LIN {X 0,Y 523.404,Z 1295.41,A -85,B 0,C 180,E1 11072.533,E2 11072.533} C_VEL
LIN {X 0,Y 523.489,Z 1283.229,A -85,B 0,C 180,E1 11079.214,E2 11079.214} C_VEL
LIN {X 0,Y 524.787,Z 1258.62,A -85,B 0,C 180,E1 11085.339,E2 11085.339} C_VEL
LIN {X 0,Y 527.688,Z 1221.289,A -85,B 0,C 180,E1 11090.919,E2 11090.919} C_VEL
LIN {X 0,Y 532.012,Z 1167.625,A -85,B 0,C 180,E1 11096.112,E2 11096.112} C_VEL
LIN {X 0,Y 537.414,Z 1096.373,A -85,B 0,C 180,E1 11100.613,E2 11100.613} C_VEL
LIN {X 0,Y 541.812,Z 1015.252,A -85,B 0,C 180,E1 11103.94,E2 11103.94} C_VEL
LIN {X 0,Y 528.076,Z 964.087,A -85,B 0,C 180,E1 11106.5,E2 11106.5} C_VEL
LIN {X 0,Y 521.805,Z 948.94,A -85,B 0,C 180,E1 11107.691,E2 11107.691} C_VEL
LIN {X 0,Y 521.684,Z 948.94,A -85,B 0,C 180,E1 11116.888,E2 11116.888} C_VEL
LIN {X 0,Y 521.742,Z 949.764,A -85,B 0,C 180,E1 11120.206,E2 11120.206} C_VEL
LIN {X 0,Y 539.683,Z 996.244,A -85,B 0,C 180,E1 11122.459,E2 11122.459} C_VEL
LIN {X 0,Y 545.905,Z 1027.625,A -85,B 0,C 180,E1 11123.887,E2 11123.887} C_VEL
LIN {X 0,Y 541.126,Z 1086.246,A -85,B 0,C 180,E1 11126.86,E2 11126.86} C_VEL
LIN {X 0,Y 534.613,Z 1139.181,A -85,B 0,C 180,E1 11131.402,E2 11131.402} C_VEL
LIN {X 0,Y 528.549,Z 1183.072,A -85,B 0,C 180,E1 11137.431,E2 11137.431} C_VEL
LIN {X 0,Y 524.596,Z 1214.168,A -85,B 0,C 180,E1 11144.494,E2 11144.494} C_VEL
LIN {X 0,Y 523.276,Z 1230.193,A -85,B 0,C 180,E1 11151.677,E2 11151.677} C_VEL
LIN {X 0,Y 523.605,Z 1232.827,A -85,B 0,C 180,E1 11159.186,E2 11159.186} C_VEL
LIN {X 0,Y 524.011,Z 1221.488,A -85,B 0,C 180,E1 11166.67,E2 11166.67} C_VEL
LIN {X 0,Y 526.252,Z 1196.329,A -85,B 0,C 180,E1 11173.782,E2 11173.782} C_VEL
LIN {X 0,Y 531.422,Z 1159.095,A -85,B 0,C 180,E1 11180.061,E2 11180.061} C_VEL
LIN {X 0,Y 538.978,Z 1108.706,A -85,B 0,C 180,E1 11185.5,E2 11185.5} C_VEL
LIN {X 0,Y 546.377,Z 1049.845,A -85,B 0,C 180,E1 11189.517,E2 11189.517} C_VEL
LIN {X 0,Y 547.74,Z 1014.319,A -85,B 0,C 180,E1 11191.228,E2 11191.228} C_VEL
LIN {X 0,Y 521.747,Z 948.94,A -85,B 0,C 180,E1 11194.949,E2 11194.949} C_VEL
LIN {X 0,Y 521.658,Z 948.94,A -85,B 0,C 180,E1 11205.49,E2 11205.49} C_VEL
LIN {X 0,Y 521.836,Z 948.94,A -85,B 0,C 180,E1 11215.411,E2 11215.411} C_VEL
LIN {X 0,Y 522.074,Z 948.94,A -85,B 0,C 180,E1 11225.032,E2 11225.032} C_VEL
LIN {X 0,Y 522.428,Z 950.12,A -85,B 0,C 180,E1 11228.088,E2 11228.088} C_VEL
LIN {X 0,Y 534.24,Z 993.796,A -85,B 0,C 180,E1 11229.217,E2 11229.217} C_VEL
LIN {X 0,Y 533.431,Z 1050.572,A -85,B 0,C 180,E1 11230.538,E2 11230.538} C_VEL
LIN {X 0,Y 530.805,Z 1095.033,A -85,B 0,C 180,E1 11233.207,E2 11233.207} C_VEL
LIN {X 0,Y 527.666,Z 1131.511,A -85,B 0,C 180,E1 11237.293,E2 11237.293} C_VEL
LIN {X 0,Y 525.494,Z 1154.569,A -85,B 0,C 180,E1 11242.076,E2 11242.076} C_VEL
LIN {X 0,Y 524.449,Z 1165.004,A -85,B 0,C 180,E1 11247.472,E2 11247.472} C_VEL
LIN {X 0,Y 524.553,Z 1161.476,A -85,B 0,C 180,E1 11253.088,E2 11253.088} C_VEL
LIN {X 0,Y 526.11,Z 1144.372,A -85,B 0,C 180,E1 11258.25,E2 11258.25} C_VEL
LIN {X 0,Y 528.756,Z 1113.784,A -85,B 0,C 180,E1 11262.808,E2 11262.808} C_VEL
LIN {X 0,Y 531.912,Z 1071.936,A -85,B 0,C 180,E1 11266.212,E2 11266.212} C_VEL
LIN {X 0,Y 533.887,Z 1023.989,A -85,B 0,C 180,E1 11268.092,E2 11268.092} C_VEL
LIN {X 0,Y 531.672,Z 981.287,A -85,B 0,C 180,E1 11268.845,E2 11268.845} C_VEL
LIN {X 0,Y 522.302,Z 948.94,A -85,B 0,C 180,E1 11269.716,E2 11269.716} C_VEL
LIN {X 0,Y 521.815,Z 948.94,A -85,B 0,C 180,E1 11278.623,E2 11278.623} C_VEL
LIN {X 0,Y 521.589,Z 948.94,A -85,B 0,C 180,E1 11288.66,E2 11288.66} C_VEL
LIN {X 0,Y 521.759,Z 948.94,A -85,B 0,C 180,E1 11297.801,E2 11297.801} C_VEL
LIN {X 0,Y 521.904,Z 948.94,A -85,B 0,C 180,E1 11307.432,E2 11307.432} C_VEL
LIN {X 0,Y 522.123,Z 948.94,A -85,B 0,C 180,E1 11316.876,E2 11316.876} C_VEL
LIN {X 0,Y 523.018,Z 948.94,A -85,B 0,C 180,E1 11327.412,E2 11327.412} C_VEL
LIN {X 0,Y 523.223,Z 948.94,A -85,B 0,C 180,E1 11337.49,E2 11337.49} C_VEL
LIN {X 0,Y 522.846,Z 948.94,A -85,B 0,C 180,E1 11345.815,E2 11345.815} C_VEL
LIN {X 0,Y 522.335,Z 948.94,A -85,B 0,C 180,E1 11354.283,E2 11354.283} C_VEL
LIN {X 0,Y 521.848,Z 948.94,A -85,B 0,C 180,E1 11363.774,E2 11363.774} C_VEL
LIN {X 0,Y 522.135,Z 948.94,A -85,B 0,C 180,E1 11372.513,E2 11372.513} C_VEL
LIN {X 0,Y 521.87,Z 948.94,A -85,B 0,C 180,E1 11382.212,E2 11382.212} C_VEL
LIN {X 0,Y 522.147,Z 950.842,A -85,B 0,C 180,E1 11389.649,E2 11389.649} C_VEL
LIN {X 0,Y 548.684,Z 1012.45,A -85,B 0,C 180,E1 11393.235,E2 11393.235} C_VEL
LIN {X 0,Y 553.607,Z 1033.275,A -85,B 0,C 180,E1 11394.277,E2 11394.277} C_VEL
LIN {X 0,Y 545.069,Z 1104.086,A -85,B 0,C 180,E1 11397.289,E2 11397.289} C_VEL
LIN {X 0,Y 536.289,Z 1168.912,A -85,B 0,C 180,E1 11401.874,E2 11401.874} C_VEL
LIN {X 0,Y 529.352,Z 1222.539,A -85,B 0,C 180,E1 11407.724,E2 11407.724} C_VEL
LIN {X 0,Y 528.996,Z 1226.369,A -85,B 0,C 180,E1 11408.252,E2 11408.252} C_VEL
LIN {X 0,Y 518.591,Z 1246.508,A -85,B 0,C 180,E1 11411.254,E2 11411.254} C_VEL
LIN {X 0,Y 515.998,Z 1275.634,A -85,B 0,C 180,E1 11417.734,E2 11417.734} C_VEL
LIN {X 0,Y 515.225,Z 1291.568,A -85,B 0,C 180,E1 11424.126,E2 11424.126} C_VEL
LIN {X 0,Y 515.63,Z 1295.874,A -85,B 0,C 180,E1 11430.885,E2 11430.885} C_VEL
LIN {X 0,Y 515.565,Z 1285.947,A -85,B 0,C 180,E1 11438.078,E2 11438.078} C_VEL
LIN {X 0,Y 516.597,Z 1262.844,A -85,B 0,C 180,E1 11444.5,E2 11444.5} C_VEL
LIN {X 0,Y 519.374,Z 1226.398,A -85,B 0,C 180,E1 11450.375,E2 11450.375} C_VEL
LIN {X 0,Y 523.644,Z 1174.489,A -85,B 0,C 180,E1 11455.732,E2 11455.732} C_VEL
LIN {X 0,Y 529.25,Z 1104.542,A -85,B 0,C 180,E1 11460.451,E2 11460.451} C_VEL
LIN {X 0,Y 534.399,Z 1016.776,A -85,B 0,C 180,E1 11464.282,E2 11464.282} C_VEL
LIN {X 0,Y 521.584,Z 967.062,A -85,B 0,C 180,E1 11466.923,E2 11466.923} C_VEL
LIN {X 0,Y 513.714,Z 948.94,A -85,B 0,C 180,E1 11468.494,E2 11468.494} C_VEL
LIN {X 0,Y 513.65,Z 948.94,A -85,B 0,C 180,E1 11478.351,E2 11478.351} C_VEL
LIN {X 0,Y 513.81,Z 950.366,A -85,B 0,C 180,E1 11479.449,E2 11479.449} C_VEL
LIN {X 0,Y 531.259,Z 991.381,A -85,B 0,C 180,E1 11481.74,E2 11481.74} C_VEL
LIN {X 0,Y 538.985,Z 1029.938,A -85,B 0,C 180,E1 11483.519,E2 11483.519} C_VEL
LIN {X 0,Y 534.021,Z 1087.732,A -85,B 0,C 180,E1 11486.506,E2 11486.506} C_VEL
LIN {X 0,Y 527.085,Z 1141.072,A -85,B 0,C 180,E1 11491.18,E2 11491.18} C_VEL
LIN {X 0,Y 520.761,Z 1184.515,A -85,B 0,C 180,E1 11497.3,E2 11497.3} C_VEL
LIN {X 0,Y 516.773,Z 1214.514,A -85,B 0,C 180,E1 11504.253,E2 11504.253} C_VEL
LIN {X 0,Y 515.315,Z 1230.656,A -85,B 0,C 180,E1 11511.562,E2 11511.562} C_VEL
LIN {X 0,Y 515.606,Z 1233.326,A -85,B 0,C 180,E1 11519.173,E2 11519.173} C_VEL
LIN {X 0,Y 516.048,Z 1221.99,A -85,B 0,C 180,E1 11526.773,E2 11526.773} C_VEL
LIN {X 0,Y 518.237,Z 1198.687,A -85,B 0,C 180,E1 11533.567,E2 11533.567} C_VEL
LIN {X 0,Y 523.43,Z 1162.578,A -85,B 0,C 180,E1 11539.938,E2 11539.938} C_VEL
LIN {X 0,Y 531.263,Z 1112.234,A -85,B 0,C 180,E1 11545.585,E2 11545.585} C_VEL
LIN {X 0,Y 538.978,Z 1052.791,A -85,B 0,C 180,E1 11549.776,E2 11549.776} C_VEL
LIN {X 0,Y 540.615,Z 1016.514,A -85,B 0,C 180,E1 11551.57,E2 11551.57} C_VEL
LIN {X 0,Y 513.896,Z 950.514,A -85,B 0,C 180,E1 11555.373,E2 11555.373} C_VEL
LIN {X 0,Y 513.611,Z 948.94,A -85,B 0,C 180,E1 11564.007,E2 11564.007} C_VEL
LIN {X 0,Y 513.748,Z 948.94,A -85,B 0,C 180,E1 11572.688,E2 11572.688} C_VEL
LIN {X 0,Y 513.949,Z 948.94,A -85,B 0,C 180,E1 11582.722,E2 11582.722} C_VEL
LIN {X 0,Y 514.309,Z 949.389,A -85,B 0,C 180,E1 11587.711,E2 11587.711} C_VEL
LIN {X 0,Y 526.783,Z 995.817,A -85,B 0,C 180,E1 11588.937,E2 11588.937} C_VEL
LIN {X 0,Y 525.933,Z 1051.308,A -85,B 0,C 180,E1 11590.252,E2 11590.252} C_VEL
LIN {X 0,Y 523.129,Z 1096.573,A -85,B 0,C 180,E1 11593.016,E2 11593.016} C_VEL
LIN {X 0,Y 519.907,Z 1132.394,A -85,B 0,C 180,E1 11597.1,E2 11597.1} C_VEL
LIN {X 0,Y 517.618,Z 1155.488,A -85,B 0,C 180,E1 11601.955,E2 11601.955} C_VEL
LIN {X 0,Y 516.53,Z 1165.949,A -85,B 0,C 180,E1 11607.433,E2 11607.433} C_VEL
LIN {X 0,Y 516.639,Z 1162.445,A -85,B 0,C 180,E1 11613.135,E2 11613.135} C_VEL
LIN {X 0,Y 518.246,Z 1145.374,A -85,B 0,C 180,E1 11618.376,E2 11618.376} C_VEL
LIN {X 0,Y 521.025,Z 1114.818,A -85,B 0,C 180,E1 11623.001,E2 11623.001} C_VEL
LIN {X 0,Y 524.299,Z 1073.62,A -85,B 0,C 180,E1 11626.42,E2 11626.42} C_VEL
LIN {X 0,Y 526.306,Z 1026.063,A -85,B 0,C 180,E1 11628.344,E2 11628.344} C_VEL
LIN {X 0,Y 524.142,Z 982.619,A -85,B 0,C 180,E1 11629.13,E2 11629.13} C_VEL
LIN {X 0,Y 514.238,Z 948.94,A -85,B 0,C 180,E1 11630.214,E2 11630.214} C_VEL
LIN {X 0,Y 513.718,Z 948.94,A -85,B 0,C 180,E1 11639.322,E2 11639.322} C_VEL
LIN {X 0,Y 513.544,Z 948.94,A -85,B 0,C 180,E1 11649.382,E2 11649.382} C_VEL
LIN {X 0,Y 513.743,Z 948.94,A -85,B 0,C 180,E1 11658.797,E2 11658.797} C_VEL
LIN {X 0,Y 513.912,Z 948.94,A -85,B 0,C 180,E1 11668.859,E2 11668.859} C_VEL
LIN {X 0,Y 514.128,Z 948.94,A -85,B 0,C 180,E1 11678.327,E2 11678.327} C_VEL
LIN {X 0,Y 515.002,Z 948.94,A -85,B 0,C 180,E1 11687.213,E2 11687.213} C_VEL
LIN {X 0,Y 515.208,Z 948.94,A -85,B 0,C 180,E1 11697.451,E2 11697.451} C_VEL
LIN {X 0,Y 514.809,Z 948.94,A -85,B 0,C 180,E1 11705.906,E2 11705.906} C_VEL
LIN {X 0,Y 514.277,Z 948.94,A -85,B 0,C 180,E1 11714.512,E2 11714.512} C_VEL
LIN {X 0,Y 513.867,Z 948.94,A -85,B 0,C 180,E1 11723.482,E2 11723.482} C_VEL
LIN {X 0,Y 514.091,Z 948.94,A -85,B 0,C 180,E1 11733.087,E2 11733.087} C_VEL
LIN {X 0,Y 513.861,Z 948.94,A -85,B 0,C 180,E1 11741.629,E2 11741.629} C_VEL
LIN {X 0,Y 514.109,Z 950.878,A -85,B 0,C 180,E1 11748.985,E2 11748.985} C_VEL
LIN {X 0,Y 540.801,Z 1011.536,A -85,B 0,C 180,E1 11752.662,E2 11752.662} C_VEL
LIN {X 0,Y 546.454,Z 1035.794,A -85,B 0,C 180,E1 11753.922,E2 11753.922} C_VEL
LIN {X 0,Y 537.589,Z 1106.059,A -85,B 0,C 180,E1 11757.018,E2 11757.018} C_VEL
LIN {X 0,Y 528.489,Z 1171.031,A -85,B 0,C 180,E1 11761.771,E2 11761.771} C_VEL
LIN {X 0,Y 521.296,Z 1224.582,A -85,B 0,C 180,E1 11767.811,E2 11767.811} C_VEL
LIN {X 0,Y 518.591,Z 1246.508,A -85,B 0,C 180,E1 11771.254,E2 11771.254} C_VEL
LIN {X 0,Y 509.389,Z 1263.5,A -85,B 0,C 180,E1 11774.581,E2 11774.581} C_VEL
LIN {X 0,Y 507.69,Z 1286.066,A -85,B 0,C 180,E1 11781.449,E2 11781.449} C_VEL
LIN {X 0,Y 507.298,Z 1294.811,A -85,B 0,C 180,E1 11787.471,E2 11787.471} C_VEL
LIN {X 0,Y 507.419,Z 1294.376,A -85,B 0,C 180,E1 11792.613,E2 11792.613} C_VEL
LIN {X 0,Y 507.528,Z 1283.01,A -85,B 0,C 180,E1 11799.073,E2 11799.073} C_VEL
LIN {X 0,Y 508.82,Z 1258.469,A -85,B 0,C 180,E1 11805.39,E2 11805.39} C_VEL
LIN {X 0,Y 511.889,Z 1220.342,A -85,B 0,C 180,E1 11811.251,E2 11811.251} C_VEL
LIN {X 0,Y 516.487,Z 1166.16,A -85,B 0,C 180,E1 11816.61,E2 11816.61} C_VEL
LIN {X 0,Y 522.8,Z 1091.128,A -85,B 0,C 180,E1 11821.45,E2 11821.45} C_VEL
LIN {X 0,Y 527.248,Z 1019.233,A -85,B 0,C 180,E1 11824.588,E2 11824.588} C_VEL
LIN {X 0,Y 515.448,Z 970.997,A -85,B 0,C 180,E1 11827.304,E2 11827.304} C_VEL
LIN {X 0,Y 505.71,Z 948.94,A -85,B 0,C 180,E1 11829.432,E2 11829.432} C_VEL
LIN {X 0,Y 505.897,Z 950.919,A -85,B 0,C 180,E1 11838.562,E2 11838.562} C_VEL
LIN {X 0,Y 522.729,Z 987.061,A -85,B 0,C 180,E1 11841.002,E2 11841.002} C_VEL
LIN {X 0,Y 532.142,Z 1031.862,A -85,B 0,C 180,E1 11843.114,E2 11843.114} C_VEL
LIN {X 0,Y 526.841,Z 1090.193,A -85,B 0,C 180,E1 11846.202,E2 11846.202} C_VEL
LIN {X 0,Y 519.561,Z 1143.117,A -85,B 0,C 180,E1 11850.962,E2 11850.962} C_VEL
LIN {X 0,Y 512.979,Z 1185.99,A -85,B 0,C 180,E1 11857.167,E2 11857.167} C_VEL
LIN {X 0,Y 508.74,Z 1216.253,A -85,B 0,C 180,E1 11864.442,E2 11864.442} C_VEL
LIN {X 0,Y 507.348,Z 1231.262,A -85,B 0,C 180,E1 11871.543,E2 11871.543} C_VEL
LIN {X 0,Y 507.622,Z 1233.825,A -85,B 0,C 180,E1 11879.16,E2 11879.16} C_VEL
LIN {X 0,Y 508.108,Z 1222.478,A -85,B 0,C 180,E1 11886.879,E2 11886.879} C_VEL
LIN {X 0,Y 510.406,Z 1199.13,A -85,B 0,C 180,E1 11893.78,E2 11893.78} C_VEL
LIN {X 0,Y 515.822,Z 1162.885,A -85,B 0,C 180,E1 11900.245,E2 11900.245} C_VEL
LIN {X 0,Y 523.934,Z 1112.633,A -85,B 0,C 180,E1 11905.942,E2 11905.942} C_VEL
LIN {X 0,Y 532.073,Z 1052.029,A -85,B 0,C 180,E1 11910.241,E2 11910.241} C_VEL
LIN {X 0,Y 533.483,Z 1018.596,A -85,B 0,C 180,E1 11911.922,E2 11911.922} C_VEL
LIN {X 0,Y 506.92,Z 953.164,A -85,B 0,C 180,E1 11915.806,E2 11915.806} C_VEL
LIN {X 0,Y 505.644,Z 948.94,A -85,B 0,C 180,E1 11916.122,E2 11916.122} C_VEL
LIN {X 0,Y 505.556,Z 948.94,A -85,B 0,C 180,E1 11925.088,E2 11925.088} C_VEL
LIN {X 0,Y 505.733,Z 948.94,A -85,B 0,C 180,E1 11934.143,E2 11934.143} C_VEL
LIN {X 0,Y 505.979,Z 948.94,A -85,B 0,C 180,E1 11944.18,E2 11944.18} C_VEL
LIN {X 0,Y 506.49,Z 950.929,A -85,B 0,C 180,E1 11947.369,E2 11947.369} C_VEL
LIN {X 0,Y 519.369,Z 998.454,A -85,B 0,C 180,E1 11948.658,E2 11948.658} C_VEL
LIN {X 0,Y 518.401,Z 1052.627,A -85,B 0,C 180,E1 11949.98,E2 11949.98} C_VEL
LIN {X 0,Y 515.44,Z 1098.32,A -85,B 0,C 180,E1 11952.838,E2 11952.838} C_VEL
LIN {X 0,Y 512.154,Z 1133.276,A -85,B 0,C 180,E1 11956.902,E2 11956.902} C_VEL
LIN {X 0,Y 509.744,Z 1156.408,A -85,B 0,C 180,E1 11961.83,E2 11961.83} C_VEL
LIN {X 0,Y 508.601,Z 1166.895,A -85,B 0,C 180,E1 11967.393,E2 11967.393} C_VEL
LIN {X 0,Y 508.687,Z 1164.568,A -85,B 0,C 180,E1 11972.522,E2 11972.522} C_VEL
LIN {X 0,Y 510.168,Z 1148.29,A -85,B 0,C 180,E1 11978.079,E2 11978.079} C_VEL
LIN {X 0,Y 512.968,Z 1119.521,A -85,B 0,C 180,E1 11982.774,E2 11982.774} C_VEL
LIN {X 0,Y 516.502,Z 1078.229,A -85,B 0,C 180,E1 11986.444,E2 11986.444} C_VEL
LIN {X 0,Y 518.704,Z 1030.52,A -85,B 0,C 180,E1 11988.546,E2 11988.546} C_VEL
LIN {X 0,Y 517.009,Z 985.389,A -85,B 0,C 180,E1 11989.385,E2 11989.385} C_VEL
LIN {X 0,Y 506.167,Z 948.94,A -85,B 0,C 180,E1 11990.593,E2 11990.593} C_VEL
LIN {X 0,Y 505.703,Z 948.94,A -85,B 0,C 180,E1 12001.164,E2 12001.164} C_VEL
LIN {X 0,Y 505.499,Z 948.94,A -85,B 0,C 180,E1 12010.135,E2 12010.135} C_VEL
LIN {X 0,Y 505.686,Z 948.94,A -85,B 0,C 180,E1 12019.851,E2 12019.851} C_VEL
LIN {X 0,Y 505.898,Z 948.94,A -85,B 0,C 180,E1 12028.652,E2 12028.652} C_VEL
LIN {X 0,Y 506.112,Z 948.94,A -85,B 0,C 180,E1 12037.966,E2 12037.966} C_VEL
LIN {X 0,Y 506.95,Z 948.94,A -85,B 0,C 180,E1 12047.006,E2 12047.006} C_VEL
LIN {X 0,Y 507.206,Z 948.94,A -85,B 0,C 180,E1 12057.41,E2 12057.41} C_VEL
LIN {X 0,Y 506.772,Z 948.94,A -85,B 0,C 180,E1 12066,E2 12066} C_VEL
LIN {X 0,Y 506.236,Z 948.94,A -85,B 0,C 180,E1 12074.747,E2 12074.747} C_VEL
LIN {X 0,Y 505.811,Z 948.94,A -85,B 0,C 180,E1 12083.913,E2 12083.913} C_VEL
LIN {X 0,Y 506.006,Z 948.94,A -85,B 0,C 180,E1 12093.685,E2 12093.685} C_VEL
LIN {X 0,Y 505.754,Z 948.94,A -85,B 0,C 180,E1 12102.755,E2 12102.755} C_VEL
LIN {X 0,Y 505.967,Z 950.512,A -85,B 0,C 180,E1 12108.28,E2 12108.28} C_VEL
LIN {X 0,Y 532.967,Z 1011.113,A -85,B 0,C 180,E1 12112.102,E2 12112.102} C_VEL
LIN {X 0,Y 539.42,Z 1037.751,A -85,B 0,C 180,E1 12113.541,E2 12113.541} C_VEL
LIN {X 0,Y 530.134,Z 1107.665,A -85,B 0,C 180,E1 12116.739,E2 12116.739} C_VEL
LIN {X 0,Y 520.604,Z 1172.989,A -85,B 0,C 180,E1 12121.66,E2 12121.66} C_VEL
LIN {X 0,Y 513.403,Z 1224.995,A -85,B 0,C 180,E1 12127.681,E2 12127.681} C_VEL
LIN {X 0,Y 509.389,Z 1263.5,A -85,B 0,C 180,E1 12134.581,E2 12134.581} C_VEL
LIN {X 0,Y 499.959,Z 1276.93,A -85,B 0,C 180,E1 12138.159,E2 12138.159} C_VEL
LIN {X 0,Y 499.373,Z 1291.79,A -85,B 0,C 180,E1 12144.813,E2 12144.813} C_VEL
LIN {X 0,Y 499.658,Z 1294.881,A -85,B 0,C 180,E1 12150.913,E2 12150.913} C_VEL
LIN {X 0,Y 499.603,Z 1285.658,A -85,B 0,C 180,E1 12157.898,E2 12157.898} C_VEL
LIN {X 0,Y 500.584,Z 1264.051,A -85,B 0,C 180,E1 12164.262,E2 12164.262} C_VEL
LIN {X 0,Y 503.346,Z 1228.365,A -85,B 0,C 180,E1 12170.328,E2 12170.328} C_VEL
LIN {X 0,Y 507.884,Z 1176.454,A -85,B 0,C 180,E1 12175.952,E2 12175.952} C_VEL
LIN {X 0,Y 514.087,Z 1104.881,A -85,B 0,C 180,E1 12181.023,E2 12181.023} C_VEL
LIN {X 0,Y 520.119,Z 1021.432,A -85,B 0,C 180,E1 12184.935,E2 12184.935} C_VEL
LIN {X 0,Y 509.447,Z 974.988,A -85,B 0,C 180,E1 12187.703,E2 12187.703} C_VEL
LIN {X 0,Y 497.611,Z 948.94,A -85,B 0,C 180,E1 12190.605,E2 12190.605} C_VEL
LIN {X 0,Y 497.832,Z 950.883,A -85,B 0,C 180,E1 12197.409,E2 12197.409} C_VEL
LIN {X 0,Y 513.079,Z 980.496,A -85,B 0,C 180,E1 12200.039,E2 12200.039} C_VEL
LIN {X 0,Y 525.402,Z 1034.002,A -85,B 0,C 180,E1 12202.698,E2 12202.698} C_VEL
LIN {X 0,Y 519.823,Z 1091.852,A -85,B 0,C 180,E1 12205.822,E2 12205.822} C_VEL
LIN {X 0,Y 512.448,Z 1143.369,A -85,B 0,C 180,E1 12210.52,E2 12210.52} C_VEL
LIN {X 0,Y 505.612,Z 1185.586,A -85,B 0,C 180,E1 12216.661,E2 12216.661} C_VEL
LIN {X 0,Y 501.196,Z 1215.295,A -85,B 0,C 180,E1 12223.75,E2 12223.75} C_VEL
LIN {X 0,Y 499.403,Z 1231.435,A -85,B 0,C 180,E1 12231.171,E2 12231.171} C_VEL
LIN {X 0,Y 499.172,Z 1234.961,A -85,B 0,C 180,E1 12237.403,E2 12237.403} C_VEL
LIN {X 0,Y 500.17,Z 1226.764,A -85,B 0,C 180,E1 12245.24,E2 12245.24} C_VEL
LIN {X 0,Y 502.045,Z 1204.991,A -85,B 0,C 180,E1 12252.679,E2 12252.679} C_VEL
LIN {X 0,Y 507.332,Z 1169.076,A -85,B 0,C 180,E1 12259.671,E2 12259.671} C_VEL
LIN {X 0,Y 515.392,Z 1120.824,A -85,B 0,C 180,E1 12265.561,E2 12265.561} C_VEL
LIN {X 0,Y 523.552,Z 1063.685,A -85,B 0,C 180,E1 12269.998,E2 12269.998} C_VEL
LIN {X 0,Y 526.397,Z 1021.071,A -85,B 0,C 180,E1 12272.256,E2 12272.256} C_VEL
LIN {X 0,Y 500.371,Z 956.509,A -85,B 0,C 180,E1 12276.197,E2 12276.197} C_VEL
LIN {X 0,Y 497.608,Z 948.94,A -85,B 0,C 180,E1 12276.857,E2 12276.857} C_VEL
LIN {X 0,Y 497.502,Z 948.94,A -85,B 0,C 180,E1 12286.611,E2 12286.611} C_VEL
LIN {X 0,Y 497.697,Z 948.94,A -85,B 0,C 180,E1 12295.616,E2 12295.616} C_VEL
LIN {X 0,Y 497.999,Z 948.94,A -85,B 0,C 180,E1 12305.666,E2 12305.666} C_VEL
LIN {X 0,Y 498.384,Z 950.661,A -85,B 0,C 180,E1 12306.974,E2 12306.974} C_VEL
LIN {X 0,Y 511.947,Z 1000.661,A -85,B 0,C 180,E1 12308.364,E2 12308.364} C_VEL
LIN {X 0,Y 510.811,Z 1055.196,A -85,B 0,C 180,E1 12309.752,E2 12309.752} C_VEL
LIN {X 0,Y 507.651,Z 1100.916,A -85,B 0,C 180,E1 12312.728,E2 12312.728} C_VEL
LIN {X 0,Y 504.214,Z 1135.547,A -85,B 0,C 180,E1 12316.913,E2 12316.913} C_VEL
LIN {X 0,Y 501.64,Z 1158.633,A -85,B 0,C 180,E1 12322.134,E2 12322.134} C_VEL
LIN {X 0,Y 500.684,Z 1167.839,A -85,B 0,C 180,E1 12327.352,E2 12327.352} C_VEL
LIN {X 0,Y 500.769,Z 1165.535,A -85,B 0,C 180,E1 12332.562,E2 12332.562} C_VEL
LIN {X 0,Y 502.31,Z 1149.285,A -85,B 0,C 180,E1 12338.206,E2 12338.206} C_VEL
LIN {X 0,Y 505.262,Z 1120.544,A -85,B 0,C 180,E1 12342.972,E2 12342.972} C_VEL
LIN {X 0,Y 508.895,Z 1080.171,A -85,B 0,C 180,E1 12346.639,E2 12346.639} C_VEL
LIN {X 0,Y 511.18,Z 1031.918,A -85,B 0,C 180,E1 12348.826,E2 12348.826} C_VEL
LIN {X 0,Y 509.457,Z 986.66,A -85,B 0,C 180,E1 12349.689,E2 12349.689} C_VEL
LIN {X 0,Y 498.126,Z 948.94,A -85,B 0,C 180,E1 12350.926,E2 12350.926} C_VEL
LIN {X 0,Y 497.652,Z 948.94,A -85,B 0,C 180,E1 12360.153,E2 12360.153} C_VEL
LIN {X 0,Y 497.437,Z 948.94,A -85,B 0,C 180,E1 12368.889,E2 12368.889} C_VEL
LIN {X 0,Y 497.59,Z 948.94,A -85,B 0,C 180,E1 12378.996,E2 12378.996} C_VEL
LIN {X 0,Y 497.777,Z 948.94,A -85,B 0,C 180,E1 12387.73,E2 12387.73} C_VEL
LIN {X 0,Y 498.119,Z 948.94,A -85,B 0,C 180,E1 12398.168,E2 12398.168} C_VEL
LIN {X 0,Y 498.929,Z 948.94,A -85,B 0,C 180,E1 12408.578,E2 12408.578} C_VEL
LIN {X 0,Y 498.723,Z 948.94,A -85,B 0,C 180,E1 12419.111,E2 12419.111} C_VEL
LIN {X 0,Y 498.4,Z 948.94,A -85,B 0,C 180,E1 12427.859,E2 12427.859} C_VEL
LIN {X 0,Y 498.018,Z 948.94,A -85,B 0,C 180,E1 12436.812,E2 12436.812} C_VEL
LIN {X 0,Y 497.807,Z 948.94,A -85,B 0,C 180,E1 12446.219,E2 12446.219} C_VEL
LIN {X 0,Y 497.961,Z 948.94,A -85,B 0,C 180,E1 12456.226,E2 12456.226} C_VEL
LIN {X 0,Y 497.632,Z 948.94,A -85,B 0,C 180,E1 12465.763,E2 12465.763} C_VEL
LIN {X 0,Y 497.873,Z 950.527,A -85,B 0,C 180,E1 12467.571,E2 12467.571} C_VEL
LIN {X 0,Y 525.392,Z 1011.487,A -85,B 0,C 180,E1 12471.576,E2 12471.576} C_VEL
LIN {X 0,Y 532.269,Z 1040.522,A -85,B 0,C 180,E1 12473.186,E2 12473.186} C_VEL
LIN {X 0,Y 522.081,Z 1112.551,A -85,B 0,C 180,E1 12476.658,E2 12476.658} C_VEL
LIN {X 0,Y 512.578,Z 1176.014,A -85,B 0,C 180,E1 12481.658,E2 12481.658} C_VEL
LIN {X 0,Y 505.232,Z 1228.38,A -85,B 0,C 180,E1 12487.997,E2 12487.997} C_VEL
LIN {X 0,Y 501.129,Z 1266.028,A -85,B 0,C 180,E1 12495.131,E2 12495.131} C_VEL
LIN {X 0,Y 499.959,Z 1276.93,A -85,B 0,C 180,E1 12498.159,E2 12498.159} C_VEL
LIN {X 0,Y 491.499,Z 1286.659,A -85,B 0,C 180,E1 12502.006,E2 12502.006} C_VEL
LIN {X 0,Y 491.341,Z 1293.818,A -85,B 0,C 180,E1 12507.389,E2 12507.389} C_VEL
LIN {X 0,Y 491.427,Z 1293.352,A -85,B 0,C 180,E1 12512.698,E2 12512.698} C_VEL
LIN {X 0,Y 491.552,Z 1282.238,A -85,B 0,C 180,E1 12519.135,E2 12519.135} C_VEL
LIN {X 0,Y 492.857,Z 1258.631,A -85,B 0,C 180,E1 12525.443,E2 12525.443} C_VEL
LIN {X 0,Y 496.003,Z 1221.043,A -85,B 0,C 180,E1 12531.43,E2 12531.43} C_VEL
LIN {X 0,Y 500.972,Z 1166.531,A -85,B 0,C 180,E1 12537.038,E2 12537.038} C_VEL
LIN {X 0,Y 507.961,Z 1091.032,A -85,B 0,C 180,E1 12542.131,E2 12542.131} C_VEL
LIN {X 0,Y 512.806,Z 1022.595,A -85,B 0,C 180,E1 12545.364,E2 12545.364} C_VEL
LIN {X 0,Y 503.338,Z 978.264,A -85,B 0,C 180,E1 12548.182,E2 12548.182} C_VEL
LIN {X 0,Y 492.001,Z 954.679,A -85,B 0,C 180,E1 12551.175,E2 12551.175} C_VEL
LIN {X 0,Y 489.505,Z 948.94,A -85,B 0,C 180,E1 12552.802,E2 12552.802} C_VEL
LIN {X 0,Y 489.846,Z 951.113,A -85,B 0,C 180,E1 12555.688,E2 12555.688} C_VEL
LIN {X 0,Y 499.324,Z 966.488,A -85,B 0,C 180,E1 12558.178,E2 12558.178} C_VEL
LIN {X 0,Y 513.048,Z 1002.641,A -85,B 0,C 180,E1 12560.54,E2 12560.54} C_VEL
LIN {X 0,Y 518.576,Z 1038.567,A -85,B 0,C 180,E1 12562.36,E2 12562.36} C_VEL
LIN {X 0,Y 512.537,Z 1096.201,A -85,B 0,C 180,E1 12565.625,E2 12565.625} C_VEL
LIN {X 0,Y 504.641,Z 1147.323,A -85,B 0,C 180,E1 12570.498,E2 12570.498} C_VEL
LIN {X 0,Y 497.553,Z 1188.625,A -85,B 0,C 180,E1 12576.798,E2 12576.798} C_VEL
LIN {X 0,Y 493.129,Z 1217.158,A -85,B 0,C 180,E1 12583.936,E2 12583.936} C_VEL
LIN {X 0,Y 491.451,Z 1231.922,A -85,B 0,C 180,E1 12591.027,E2 12591.027} C_VEL
